(* Logix 5000 project; controller QW361 vendor 1 type 14 code 107 rev 32.11; software revision 32.00; part 10 of 20 *)

        [1241].log_data[0].time := 300.0, [1241].log_data[0].minminute := 55, [1241].log_data[0].maxminute := 55, [1241].log_data[0].valid := 1, [1241].log_data[1].valid := 1, [1241].log_data[2].valid := 1, [1241].log_data[3].valid := 1, [1241].log_data[4].valid := 1, [1241].time.Year := 2022, [1241].time.Month := 4, [1241].time.Day := 28, [1241].time.Hour := 4, [1241].time.Minute := 59, [1241].time.Second := 59, [1241].time.DST_ON := 1, [1242].log_data[0].min := 1.0, [1242].log_data[0].max := 1.0, [1242].log_data[0].total := 300.0, [1242].log_data[0].time := 300.0, [1242].log_data[0].valid := 1, [1242].log_data[1].valid := 1, [1242].log_data[2].valid := 1, [1242].log_data[3].valid := 1, [1242].log_data[4].valid := 1, [1242].time.Year := 2022, [1242].time.Month := 4, [1242].time.Day := 28, [1242].time.Hour := 5, [1242].time.Minute := 4, [1242].time.Second := 59, [1242].time.DST_ON := 1, [1243].log_data[0].min := 1.0, [1243].log_data[0].max := 1.0, [1243].log_data[0].total := 300.0, [1243].log_data[0].time := 300.0, [1243].log_data[0].minminute := 5, [1243].log_data[0].maxminute := 5, [1243].log_data[0].valid := 1, [1243].log_data[1].valid := 1, [1243].log_data[2].valid := 1, [1243].log_data[3].valid := 1, [1243].log_data[4].valid := 1, [1243].time.Year := 2022, [1243].time.Month := 4, [1243].time.Day := 28, [1243].time.Hour := 5, [1243].time.Minute := 9, [1243].time.Second := 59, [1243].time.DST_ON := 1, [1244].log_data[0].min := 1.0, [1244].log_data[0].max := 1.0, [1244].log_data[0].total := 300.0, [1244].log_data[0].time := 300.0, [1244].log_data[0].minminute := 10, [1244].log_data[0].maxminute := 10, [1244].log_data[0].valid := 1, [1244].log_data[1].valid := 1, [1244].log_data[2].valid := 1, [1244].log_data[3].valid := 1, [1244].log_data[4].valid := 1,
        [1244].time.Year := 2022, [1244].time.Month := 4, [1244].time.Day := 28, [1244].time.Hour := 5, [1244].time.Minute := 14, [1244].time.Second := 59, [1244].time.DST_ON := 1, [1245].log_data[0].min := 1.0, [1245].log_data[0].max := 1.0, [1245].log_data[0].total := 300.0, [1245].log_data[0].time := 300.0, [1245].log_data[0].minminute := 15, [1245].log_data[0].maxminute := 15, [1245].log_data[0].valid := 1, [1245].log_data[1].valid := 1, [1245].log_data[2].valid := 1, [1245].log_data[3].valid := 1, [1245].log_data[4].valid := 1, [1245].time.Year := 2022, [1245].time.Month := 4, [1245].time.Day := 28, [1245].time.Hour := 5, [1245].time.Minute := 19, [1245].time.Second := 59, [1245].time.DST_ON := 1, [1246].log_data[0].min := 1.0, [1246].log_data[0].max := 1.0, [1246].log_data[0].total := 300.0, [1246].log_data[0].time := 300.0, [1246].log_data[0].minminute := 20, [1246].log_data[0].maxminute := 20, [1246].log_data[0].valid := 1, [1246].log_data[1].valid := 1, [1246].log_data[2].valid := 1, [1246].log_data[3].valid := 1, [1246].log_data[4].valid := 1, [1246].time.Year := 2022, [1246].time.Month := 4, [1246].time.Day := 28, [1246].time.Hour := 5, [1246].time.Minute := 24, [1246].time.Second := 59, [1246].time.DST_ON := 1, [1247].log_data[0].min := 1.0, [1247].log_data[0].max := 1.0, [1247].log_data[0].total := 300.0, [1247].log_data[0].time := 300.0, [1247].log_data[0].minminute := 25, [1247].log_data[0].maxminute := 25, [1247].log_data[0].valid := 1, [1247].log_data[1].valid := 1, [1247].log_data[2].valid := 1, [1247].log_data[3].valid := 1, [1247].log_data[4].valid := 1, [1247].time.Year := 2022, [1247].time.Month := 4, [1247].time.Day := 28, [1247].time.Hour := 5, [1247].time.Minute := 29, [1247].time.Second := 59,
        [1247].time.DST_ON := 1, [1248].log_data[0].min := 1.0, [1248].log_data[0].max := 1.0, [1248].log_data[0].total := 300.0, [1248].log_data[0].time := 300.0, [1248].log_data[0].minminute := 30, [1248].log_data[0].maxminute := 30, [1248].log_data[0].valid := 1, [1248].log_data[1].valid := 1, [1248].log_data[2].valid := 1, [1248].log_data[3].valid := 1, [1248].log_data[4].valid := 1, [1248].time.Year := 2022, [1248].time.Month := 4, [1248].time.Day := 28, [1248].time.Hour := 5, [1248].time.Minute := 34, [1248].time.Second := 59, [1248].time.DST_ON := 1, [1249].log_data[0].min := 1.0, [1249].log_data[0].max := 1.0, [1249].log_data[0].total := 300.0, [1249].log_data[0].time := 300.0, [1249].log_data[0].minminute := 35, [1249].log_data[0].maxminute := 35, [1249].log_data[0].valid := 1, [1249].log_data[1].valid := 1, [1249].log_data[2].valid := 1, [1249].log_data[3].valid := 1, [1249].log_data[4].valid := 1, [1249].time.Year := 2022, [1249].time.Month := 4, [1249].time.Day := 28, [1249].time.Hour := 5, [1249].time.Minute := 39, [1249].time.Second := 59, [1249].time.DST_ON := 1, [1250].log_data[0].min := 1.0, [1250].log_data[0].max := 1.0, [1250].log_data[0].total := 300.0, [1250].log_data[0].time := 300.0, [1250].log_data[0].minminute := 40, [1250].log_data[0].maxminute := 40, [1250].log_data[0].valid := 1, [1250].log_data[1].valid := 1, [1250].log_data[2].valid := 1, [1250].log_data[3].valid := 1, [1250].log_data[4].valid := 1, [1250].time.Year := 2022, [1250].time.Month := 4, [1250].time.Day := 28, [1250].time.Hour := 5, [1250].time.Minute := 44, [1250].time.Second := 59, [1250].time.DST_ON := 1, [1251].log_data[0].min := 1.0, [1251].log_data[0].max := 1.0, [1251].log_data[0].total := 300.0, [1251].log_data[0].time := 300.0, [1251].log_data[0].minminute := 45,
        [1251].log_data[0].maxminute := 45, [1251].log_data[0].valid := 1, [1251].log_data[1].valid := 1, [1251].log_data[2].valid := 1, [1251].log_data[3].valid := 1, [1251].log_data[4].valid := 1, [1251].time.Year := 2022, [1251].time.Month := 4, [1251].time.Day := 28, [1251].time.Hour := 5, [1251].time.Minute := 49, [1251].time.Second := 59, [1251].time.DST_ON := 1, [1252].log_data[0].min := 1.0, [1252].log_data[0].max := 1.0, [1252].log_data[0].total := 300.0, [1252].log_data[0].time := 300.0, [1252].log_data[0].minminute := 50, [1252].log_data[0].maxminute := 50, [1252].log_data[0].valid := 1, [1252].log_data[1].valid := 1, [1252].log_data[2].valid := 1, [1252].log_data[3].valid := 1, [1252].log_data[4].valid := 1, [1252].time.Year := 2022, [1252].time.Month := 4, [1252].time.Day := 28, [1252].time.Hour := 5, [1252].time.Minute := 54, [1252].time.Second := 59, [1252].time.DST_ON := 1, [1253].log_data[0].min := 1.0, [1253].log_data[0].max := 1.0, [1253].log_data[0].total := 300.0, [1253].log_data[0].time := 300.0, [1253].log_data[0].minminute := 55, [1253].log_data[0].maxminute := 55, [1253].log_data[0].valid := 1, [1253].log_data[1].valid := 1, [1253].log_data[2].valid := 1, [1253].log_data[3].valid := 1, [1253].log_data[4].valid := 1, [1253].time.Year := 2022, [1253].time.Month := 4, [1253].time.Day := 28, [1253].time.Hour := 5, [1253].time.Minute := 59, [1253].time.Second := 59, [1253].time.DST_ON := 1, [1254].log_data[0].min := 1.0, [1254].log_data[0].max := 1.0, [1254].log_data[0].total := 300.0, [1254].log_data[0].time := 300.0, [1254].log_data[0].valid := 1, [1254].log_data[1].valid := 1, [1254].log_data[2].valid := 1, [1254].log_data[3].valid := 1, [1254].log_data[4].valid := 1, [1254].time.Year := 2022, [1254].time.Month := 4,
        [1254].time.Day := 28, [1254].time.Hour := 6, [1254].time.Minute := 4, [1254].time.Second := 59, [1254].time.DST_ON := 1, [1255].log_data[0].min := 1.0, [1255].log_data[0].max := 1.0, [1255].log_data[0].total := 300.0, [1255].log_data[0].time := 300.0, [1255].log_data[0].minminute := 5, [1255].log_data[0].maxminute := 5, [1255].log_data[0].valid := 1, [1255].log_data[1].valid := 1, [1255].log_data[2].valid := 1, [1255].log_data[3].valid := 1, [1255].log_data[4].valid := 1, [1255].time.Year := 2022, [1255].time.Month := 4, [1255].time.Day := 28, [1255].time.Hour := 6, [1255].time.Minute := 9, [1255].time.Second := 59, [1255].time.DST_ON := 1, [1256].log_data[0].min := 1.0, [1256].log_data[0].max := 1.0, [1256].log_data[0].total := 300.0, [1256].log_data[0].time := 300.0, [1256].log_data[0].minminute := 10, [1256].log_data[0].maxminute := 10, [1256].log_data[0].valid := 1, [1256].log_data[1].valid := 1, [1256].log_data[2].valid := 1, [1256].log_data[3].valid := 1, [1256].log_data[4].valid := 1, [1256].time.Year := 2022, [1256].time.Month := 4, [1256].time.Day := 28, [1256].time.Hour := 6, [1256].time.Minute := 14, [1256].time.Second := 59, [1256].time.DST_ON := 1, [1257].log_data[0].min := 1.0, [1257].log_data[0].max := 1.0, [1257].log_data[0].total := 299.999, [1257].log_data[0].time := 299.999, [1257].log_data[0].minminute := 15, [1257].log_data[0].maxminute := 15, [1257].log_data[0].valid := 1, [1257].log_data[1].valid := 1, [1257].log_data[2].valid := 1, [1257].log_data[3].valid := 1, [1257].log_data[4].valid := 1, [1257].time.Year := 2022, [1257].time.Month := 4, [1257].time.Day := 28, [1257].time.Hour := 6, [1257].time.Minute := 19, [1257].time.Second := 59, [1257].time.DST_ON := 1, [1258].log_data[0].min := 1.0,
        [1258].log_data[0].max := 1.0, [1258].log_data[0].total := 300.0, [1258].log_data[0].time := 300.0, [1258].log_data[0].minminute := 20, [1258].log_data[0].maxminute := 20, [1258].log_data[0].valid := 1, [1258].log_data[1].valid := 1, [1258].log_data[2].valid := 1, [1258].log_data[3].valid := 1, [1258].log_data[4].valid := 1, [1258].time.Year := 2022, [1258].time.Month := 4, [1258].time.Day := 28, [1258].time.Hour := 6, [1258].time.Minute := 24, [1258].time.Second := 59, [1258].time.DST_ON := 1, [1259].log_data[0].min := 1.0, [1259].log_data[0].max := 1.0, [1259].log_data[0].total := 300.0, [1259].log_data[0].time := 300.0, [1259].log_data[0].minminute := 25, [1259].log_data[0].maxminute := 25, [1259].log_data[0].valid := 1, [1259].log_data[1].valid := 1, [1259].log_data[2].valid := 1, [1259].log_data[3].valid := 1, [1259].log_data[4].valid := 1, [1259].time.Year := 2022, [1259].time.Month := 4, [1259].time.Day := 28, [1259].time.Hour := 6, [1259].time.Minute := 29, [1259].time.Second := 59, [1259].time.DST_ON := 1, [1260].log_data[0].min := 1.0, [1260].log_data[0].max := 1.0, [1260].log_data[0].total := 300.0, [1260].log_data[0].time := 300.0, [1260].log_data[0].minminute := 30, [1260].log_data[0].maxminute := 30, [1260].log_data[0].valid := 1, [1260].log_data[1].valid := 1, [1260].log_data[2].valid := 1, [1260].log_data[3].valid := 1, [1260].log_data[4].valid := 1, [1260].time.Year := 2022, [1260].time.Month := 4, [1260].time.Day := 28, [1260].time.Hour := 6, [1260].time.Minute := 34, [1260].time.Second := 59, [1260].time.DST_ON := 1, [1261].log_data[0].min := 1.0, [1261].log_data[0].max := 1.0, [1261].log_data[0].total := 300.0, [1261].log_data[0].time := 300.0, [1261].log_data[0].minminute := 35, [1261].log_data[0].maxminute := 35, [1261].log_data[0].valid := 1,
        [1261].log_data[1].valid := 1, [1261].log_data[2].valid := 1, [1261].log_data[3].valid := 1, [1261].log_data[4].valid := 1, [1261].time.Year := 2022, [1261].time.Month := 4, [1261].time.Day := 28, [1261].time.Hour := 6, [1261].time.Minute := 39, [1261].time.Second := 59, [1261].time.DST_ON := 1, [1262].log_data[0].min := 1.0, [1262].log_data[0].max := 1.0, [1262].log_data[0].total := 300.0, [1262].log_data[0].time := 300.0, [1262].log_data[0].minminute := 40, [1262].log_data[0].maxminute := 40, [1262].log_data[0].valid := 1, [1262].log_data[1].valid := 1, [1262].log_data[2].valid := 1, [1262].log_data[3].valid := 1, [1262].log_data[4].valid := 1, [1262].time.Year := 2022, [1262].time.Month := 4, [1262].time.Day := 28, [1262].time.Hour := 6, [1262].time.Minute := 44, [1262].time.Second := 59, [1262].time.DST_ON := 1, [1263].log_data[0].min := 1.0, [1263].log_data[0].max := 1.0, [1263].log_data[0].total := 300.0, [1263].log_data[0].time := 300.0, [1263].log_data[0].minminute := 45, [1263].log_data[0].maxminute := 45, [1263].log_data[0].valid := 1, [1263].log_data[1].valid := 1, [1263].log_data[2].valid := 1, [1263].log_data[3].valid := 1, [1263].log_data[4].valid := 1, [1263].time.Year := 2022, [1263].time.Month := 4, [1263].time.Day := 28, [1263].time.Hour := 6, [1263].time.Minute := 49, [1263].time.Second := 59, [1263].time.DST_ON := 1, [1264].log_data[0].min := 1.0, [1264].log_data[0].max := 1.0, [1264].log_data[0].total := 300.0, [1264].log_data[0].time := 300.0, [1264].log_data[0].minminute := 50, [1264].log_data[0].maxminute := 50, [1264].log_data[0].valid := 1, [1264].log_data[1].valid := 1, [1264].log_data[2].valid := 1, [1264].log_data[3].valid := 1, [1264].log_data[4].valid := 1, [1264].time.Year := 2022, [1264].time.Month := 4,
        [1264].time.Day := 28, [1264].time.Hour := 6, [1264].time.Minute := 54, [1264].time.Second := 59, [1264].time.DST_ON := 1, [1265].log_data[0].min := 1.0, [1265].log_data[0].max := 1.0, [1265].log_data[0].total := 300.0, [1265].log_data[0].time := 300.0, [1265].log_data[0].minminute := 55, [1265].log_data[0].maxminute := 55, [1265].log_data[0].valid := 1, [1265].log_data[1].valid := 1, [1265].log_data[2].valid := 1, [1265].log_data[3].valid := 1, [1265].log_data[4].valid := 1, [1265].time.Year := 2022, [1265].time.Month := 4, [1265].time.Day := 28, [1265].time.Hour := 6, [1265].time.Minute := 59, [1265].time.Second := 59, [1265].time.DST_ON := 1, [1266].log_data[0].min := 1.0, [1266].log_data[0].max := 1.0, [1266].log_data[0].total := 300.0, [1266].log_data[0].time := 300.0, [1266].log_data[0].valid := 1, [1266].log_data[1].valid := 1, [1266].log_data[2].valid := 1, [1266].log_data[3].valid := 1, [1266].log_data[4].valid := 1, [1266].time.Year := 2022, [1266].time.Month := 4, [1266].time.Day := 28, [1266].time.Hour := 7, [1266].time.Minute := 4, [1266].time.Second := 59, [1266].time.DST_ON := 1, [1267].log_data[0].min := 1.0, [1267].log_data[0].max := 1.0, [1267].log_data[0].total := 300.0, [1267].log_data[0].time := 300.0, [1267].log_data[0].minminute := 5, [1267].log_data[0].maxminute := 5, [1267].log_data[0].valid := 1, [1267].log_data[1].valid := 1, [1267].log_data[2].valid := 1, [1267].log_data[3].valid := 1, [1267].log_data[4].valid := 1, [1267].time.Year := 2022, [1267].time.Month := 4, [1267].time.Day := 28, [1267].time.Hour := 7, [1267].time.Minute := 9, [1267].time.Second := 59, [1267].time.DST_ON := 1, [1268].log_data[0].min := 1.0, [1268].log_data[0].max := 1.0, [1268].log_data[0].total := 300.0,
        [1268].log_data[0].time := 300.0, [1268].log_data[0].minminute := 10, [1268].log_data[0].maxminute := 10, [1268].log_data[0].valid := 1, [1268].log_data[1].valid := 1, [1268].log_data[2].valid := 1, [1268].log_data[3].valid := 1, [1268].log_data[4].valid := 1, [1268].time.Year := 2022, [1268].time.Month := 4, [1268].time.Day := 28, [1268].time.Hour := 7, [1268].time.Minute := 14, [1268].time.Second := 59, [1268].time.DST_ON := 1, [1269].log_data[0].min := 1.0, [1269].log_data[0].max := 1.0, [1269].log_data[0].total := 300.0, [1269].log_data[0].time := 300.0, [1269].log_data[0].minminute := 15, [1269].log_data[0].maxminute := 15, [1269].log_data[0].valid := 1, [1269].log_data[1].valid := 1, [1269].log_data[2].valid := 1, [1269].log_data[3].valid := 1, [1269].log_data[4].valid := 1, [1269].time.Year := 2022, [1269].time.Month := 4, [1269].time.Day := 28, [1269].time.Hour := 7, [1269].time.Minute := 19, [1269].time.Second := 59, [1269].time.DST_ON := 1, [1270].log_data[0].min := 1.0, [1270].log_data[0].max := 1.0, [1270].log_data[0].total := 300.0, [1270].log_data[0].time := 300.0, [1270].log_data[0].minminute := 20, [1270].log_data[0].maxminute := 20, [1270].log_data[0].valid := 1, [1270].log_data[1].valid := 1, [1270].log_data[2].valid := 1, [1270].log_data[3].valid := 1, [1270].log_data[4].valid := 1, [1270].time.Year := 2022, [1270].time.Month := 4, [1270].time.Day := 28, [1270].time.Hour := 7, [1270].time.Minute := 24, [1270].time.Second := 59, [1270].time.DST_ON := 1, [1271].log_data[0].min := 1.0, [1271].log_data[0].max := 1.0, [1271].log_data[0].total := 300.0, [1271].log_data[0].time := 300.0, [1271].log_data[0].minminute := 25, [1271].log_data[0].maxminute := 25, [1271].log_data[0].valid := 1, [1271].log_data[1].valid := 1, [1271].log_data[2].valid := 1,
        [1271].log_data[3].valid := 1, [1271].log_data[4].valid := 1, [1271].time.Year := 2022, [1271].time.Month := 4, [1271].time.Day := 28, [1271].time.Hour := 7, [1271].time.Minute := 29, [1271].time.Second := 59, [1271].time.DST_ON := 1, [1272].log_data[0].min := 1.0, [1272].log_data[0].max := 1.0, [1272].log_data[0].total := 300.0, [1272].log_data[0].time := 300.0, [1272].log_data[0].minminute := 30, [1272].log_data[0].maxminute := 30, [1272].log_data[0].valid := 1, [1272].log_data[1].valid := 1, [1272].log_data[2].valid := 1, [1272].log_data[3].valid := 1, [1272].log_data[4].valid := 1, [1272].time.Year := 2022, [1272].time.Month := 4, [1272].time.Day := 28, [1272].time.Hour := 7, [1272].time.Minute := 34, [1272].time.Second := 59, [1272].time.DST_ON := 1, [1273].log_data[0].min := 1.0, [1273].log_data[0].max := 1.0, [1273].log_data[0].total := 300.0, [1273].log_data[0].time := 300.0, [1273].log_data[0].minminute := 35, [1273].log_data[0].maxminute := 35, [1273].log_data[0].valid := 1, [1273].log_data[1].valid := 1, [1273].log_data[2].valid := 1, [1273].log_data[3].valid := 1, [1273].log_data[4].valid := 1, [1273].time.Year := 2022, [1273].time.Month := 4, [1273].time.Day := 28, [1273].time.Hour := 7, [1273].time.Minute := 39, [1273].time.Second := 59, [1273].time.DST_ON := 1, [1274].log_data[0].min := 1.0, [1274].log_data[0].max := 1.0, [1274].log_data[0].total := 300.0, [1274].log_data[0].time := 300.0, [1274].log_data[0].minminute := 40, [1274].log_data[0].maxminute := 40, [1274].log_data[0].valid := 1, [1274].log_data[1].valid := 1, [1274].log_data[2].valid := 1, [1274].log_data[3].valid := 1, [1274].log_data[4].valid := 1, [1274].time.Year := 2022, [1274].time.Month := 4, [1274].time.Day := 28, [1274].time.Hour := 7,
        [1274].time.Minute := 44, [1274].time.Second := 59, [1274].time.DST_ON := 1, [1275].log_data[0].min := 1.0, [1275].log_data[0].max := 1.0, [1275].log_data[0].total := 300.0, [1275].log_data[0].time := 300.0, [1275].log_data[0].minminute := 45, [1275].log_data[0].maxminute := 45, [1275].log_data[0].valid := 1, [1275].log_data[1].valid := 1, [1275].log_data[2].valid := 1, [1275].log_data[3].valid := 1, [1275].log_data[4].valid := 1, [1275].time.Year := 2022, [1275].time.Month := 4, [1275].time.Day := 28, [1275].time.Hour := 7, [1275].time.Minute := 49, [1275].time.Second := 59, [1275].time.DST_ON := 1, [1276].log_data[0].min := 1.0, [1276].log_data[0].max := 1.0, [1276].log_data[0].total := 300.0, [1276].log_data[0].time := 300.0, [1276].log_data[0].minminute := 50, [1276].log_data[0].maxminute := 50, [1276].log_data[0].valid := 1, [1276].log_data[1].valid := 1, [1276].log_data[2].valid := 1, [1276].log_data[3].valid := 1, [1276].log_data[4].valid := 1, [1276].time.Year := 2022, [1276].time.Month := 4, [1276].time.Day := 28, [1276].time.Hour := 7, [1276].time.Minute := 54, [1276].time.Second := 59, [1276].time.DST_ON := 1, [1277].log_data[0].min := 1.0, [1277].log_data[0].max := 1.0, [1277].log_data[0].total := 300.0, [1277].log_data[0].time := 300.0, [1277].log_data[0].minminute := 55, [1277].log_data[0].maxminute := 55, [1277].log_data[0].valid := 1, [1277].log_data[1].valid := 1, [1277].log_data[2].valid := 1, [1277].log_data[3].valid := 1, [1277].log_data[4].valid := 1, [1277].time.Year := 2022, [1277].time.Month := 4, [1277].time.Day := 28, [1277].time.Hour := 7, [1277].time.Minute := 59, [1277].time.Second := 59, [1277].time.DST_ON := 1, [1278].log_data[0].min := 1.0, [1278].log_data[0].max := 1.0, [1278].log_data[0].total := 300.0,
        [1278].log_data[0].time := 300.0, [1278].log_data[0].valid := 1, [1278].log_data[1].valid := 1, [1278].log_data[2].valid := 1, [1278].log_data[3].valid := 1, [1278].log_data[4].valid := 1, [1278].time.Year := 2022, [1278].time.Month := 4, [1278].time.Day := 28, [1278].time.Hour := 8, [1278].time.Minute := 4, [1278].time.Second := 59, [1278].time.DST_ON := 1, [1279].log_data[0].min := 1.0, [1279].log_data[0].max := 1.0, [1279].log_data[0].total := 300.0, [1279].log_data[0].time := 300.0, [1279].log_data[0].minminute := 5, [1279].log_data[0].maxminute := 5, [1279].log_data[0].valid := 1, [1279].log_data[1].valid := 1, [1279].log_data[2].valid := 1, [1279].log_data[3].valid := 1, [1279].log_data[4].valid := 1, [1279].time.Year := 2022, [1279].time.Month := 4, [1279].time.Day := 28, [1279].time.Hour := 8, [1279].time.Minute := 9, [1279].time.Second := 59, [1279].time.DST_ON := 1, [1280].log_data[0].min := 1.0, [1280].log_data[0].max := 1.0, [1280].log_data[0].total := 300.0, [1280].log_data[0].time := 300.0, [1280].log_data[0].minminute := 10, [1280].log_data[0].maxminute := 10, [1280].log_data[0].valid := 1, [1280].log_data[1].valid := 1, [1280].log_data[2].valid := 1, [1280].log_data[3].valid := 1, [1280].log_data[4].valid := 1, [1280].time.Year := 2022, [1280].time.Month := 4, [1280].time.Day := 28, [1280].time.Hour := 8, [1280].time.Minute := 14, [1280].time.Second := 59, [1280].time.DST_ON := 1, [1281].log_data[0].min := 1.0, [1281].log_data[0].max := 1.0, [1281].log_data[0].total := 300.0, [1281].log_data[0].time := 300.0, [1281].log_data[0].minminute := 15, [1281].log_data[0].maxminute := 15, [1281].log_data[0].valid := 1, [1281].log_data[1].valid := 1, [1281].log_data[2].valid := 1, [1281].log_data[3].valid := 1, [1281].log_data[4].valid := 1,
        [1281].time.Year := 2022, [1281].time.Month := 4, [1281].time.Day := 28, [1281].time.Hour := 8, [1281].time.Minute := 19, [1281].time.Second := 59, [1281].time.DST_ON := 1, [1282].log_data[0].min := 1.0, [1282].log_data[0].max := 1.0, [1282].log_data[0].total := 300.0, [1282].log_data[0].time := 300.0, [1282].log_data[0].minminute := 20, [1282].log_data[0].maxminute := 20, [1282].log_data[0].valid := 1, [1282].log_data[1].valid := 1, [1282].log_data[2].valid := 1, [1282].log_data[3].valid := 1, [1282].log_data[4].valid := 1, [1282].time.Year := 2022, [1282].time.Month := 4, [1282].time.Day := 28, [1282].time.Hour := 8, [1282].time.Minute := 24, [1282].time.Second := 59, [1282].time.DST_ON := 1, [1283].log_data[0].min := 1.0, [1283].log_data[0].max := 1.0, [1283].log_data[0].total := 300.0, [1283].log_data[0].time := 300.0, [1283].log_data[0].minminute := 25, [1283].log_data[0].maxminute := 25, [1283].log_data[0].valid := 1, [1283].log_data[1].valid := 1, [1283].log_data[2].valid := 1, [1283].log_data[3].valid := 1, [1283].log_data[4].valid := 1, [1283].time.Year := 2022, [1283].time.Month := 4, [1283].time.Day := 28, [1283].time.Hour := 8, [1283].time.Minute := 29, [1283].time.Second := 59, [1283].time.DST_ON := 1, [1284].log_data[0].min := 1.0, [1284].log_data[0].max := 1.0, [1284].log_data[0].total := 300.0, [1284].log_data[0].time := 300.0, [1284].log_data[0].minminute := 30, [1284].log_data[0].maxminute := 30, [1284].log_data[0].valid := 1, [1284].log_data[1].valid := 1, [1284].log_data[2].valid := 1, [1284].log_data[3].valid := 1, [1284].log_data[4].valid := 1, [1284].time.Year := 2022, [1284].time.Month := 4, [1284].time.Day := 28, [1284].time.Hour := 8, [1284].time.Minute := 34, [1284].time.Second := 59,
        [1284].time.DST_ON := 1, [1285].log_data[0].min := 1.0, [1285].log_data[0].max := 1.0, [1285].log_data[0].total := 300.0, [1285].log_data[0].time := 300.0, [1285].log_data[0].minminute := 35, [1285].log_data[0].maxminute := 35, [1285].log_data[0].valid := 1, [1285].log_data[1].valid := 1, [1285].log_data[2].valid := 1, [1285].log_data[3].valid := 1, [1285].log_data[4].valid := 1, [1285].time.Year := 2022, [1285].time.Month := 4, [1285].time.Day := 28, [1285].time.Hour := 8, [1285].time.Minute := 39, [1285].time.Second := 59, [1285].time.DST_ON := 1, [1286].log_data[0].min := 1.0, [1286].log_data[0].max := 1.0, [1286].log_data[0].total := 300.0, [1286].log_data[0].time := 300.0, [1286].log_data[0].minminute := 40, [1286].log_data[0].maxminute := 40, [1286].log_data[0].valid := 1, [1286].log_data[1].valid := 1, [1286].log_data[2].valid := 1, [1286].log_data[3].valid := 1, [1286].log_data[4].valid := 1, [1286].time.Year := 2022, [1286].time.Month := 4, [1286].time.Day := 28, [1286].time.Hour := 8, [1286].time.Minute := 44, [1286].time.Second := 59, [1286].time.DST_ON := 1, [1287].log_data[0].min := 1.0, [1287].log_data[0].max := 1.0, [1287].log_data[0].total := 300.0, [1287].log_data[0].time := 300.0, [1287].log_data[0].minminute := 45, [1287].log_data[0].maxminute := 45, [1287].log_data[0].valid := 1, [1287].log_data[1].valid := 1, [1287].log_data[2].valid := 1, [1287].log_data[3].valid := 1, [1287].log_data[4].valid := 1, [1287].time.Year := 2022, [1287].time.Month := 4, [1287].time.Day := 28, [1287].time.Hour := 8, [1287].time.Minute := 49, [1287].time.Second := 59, [1287].time.DST_ON := 1, [1288].log_data[0].min := 1.0, [1288].log_data[0].max := 1.0, [1288].log_data[0].total := 300.0, [1288].log_data[0].time := 300.0, [1288].log_data[0].minminute := 50,
        [1288].log_data[0].maxminute := 50, [1288].log_data[0].valid := 1, [1288].log_data[1].valid := 1, [1288].log_data[2].valid := 1, [1288].log_data[3].valid := 1, [1288].log_data[4].valid := 1, [1288].time.Year := 2022, [1288].time.Month := 4, [1288].time.Day := 28, [1288].time.Hour := 8, [1288].time.Minute := 54, [1288].time.Second := 59, [1288].time.DST_ON := 1, [1289].log_data[0].min := 1.0, [1289].log_data[0].max := 1.0, [1289].log_data[0].total := 300.0, [1289].log_data[0].time := 300.0, [1289].log_data[0].minminute := 55, [1289].log_data[0].maxminute := 55, [1289].log_data[0].valid := 1, [1289].log_data[1].valid := 1, [1289].log_data[2].valid := 1, [1289].log_data[3].valid := 1, [1289].log_data[4].valid := 1, [1289].time.Year := 2022, [1289].time.Month := 4, [1289].time.Day := 28, [1289].time.Hour := 8, [1289].time.Minute := 59, [1289].time.Second := 59, [1289].time.DST_ON := 1, [1290].log_data[0].min := 1.0, [1290].log_data[0].max := 1.0, [1290].log_data[0].total := 300.0, [1290].log_data[0].time := 300.0, [1290].log_data[0].valid := 1, [1290].log_data[1].valid := 1, [1290].log_data[2].valid := 1, [1290].log_data[3].valid := 1, [1290].log_data[4].valid := 1, [1290].time.Year := 2022, [1290].time.Month := 4, [1290].time.Day := 28, [1290].time.Hour := 9, [1290].time.Minute := 4, [1290].time.Second := 59, [1290].time.DST_ON := 1, [1291].log_data[0].min := 1.0, [1291].log_data[0].max := 1.0, [1291].log_data[0].total := 300.0, [1291].log_data[0].time := 300.0, [1291].log_data[0].minminute := 5, [1291].log_data[0].maxminute := 5, [1291].log_data[0].valid := 1, [1291].log_data[1].valid := 1, [1291].log_data[2].valid := 1, [1291].log_data[3].valid := 1, [1291].log_data[4].valid := 1, [1291].time.Year := 2022, [1291].time.Month := 4,
        [1291].time.Day := 28, [1291].time.Hour := 9, [1291].time.Minute := 9, [1291].time.Second := 59, [1291].time.DST_ON := 1, [1292].log_data[0].min := 1.0, [1292].log_data[0].max := 1.0, [1292].log_data[0].total := 300.0, [1292].log_data[0].time := 300.0, [1292].log_data[0].minminute := 10, [1292].log_data[0].maxminute := 10, [1292].log_data[0].valid := 1, [1292].log_data[1].valid := 1, [1292].log_data[2].valid := 1, [1292].log_data[3].valid := 1, [1292].log_data[4].valid := 1, [1292].time.Year := 2022, [1292].time.Month := 4, [1292].time.Day := 28, [1292].time.Hour := 9, [1292].time.Minute := 14, [1292].time.Second := 59, [1292].time.DST_ON := 1, [1293].log_data[0].min := 1.0, [1293].log_data[0].max := 1.0, [1293].log_data[0].total := 300.0, [1293].log_data[0].time := 300.0, [1293].log_data[0].minminute := 15, [1293].log_data[0].maxminute := 15, [1293].log_data[0].valid := 1, [1293].log_data[1].valid := 1, [1293].log_data[2].valid := 1, [1293].log_data[3].valid := 1, [1293].log_data[4].valid := 1, [1293].time.Year := 2022, [1293].time.Month := 4, [1293].time.Day := 28, [1293].time.Hour := 9, [1293].time.Minute := 19, [1293].time.Second := 59, [1293].time.DST_ON := 1, [1294].log_data[0].min := 1.0, [1294].log_data[0].max := 1.0, [1294].log_data[0].total := 300.0, [1294].log_data[0].time := 300.0, [1294].log_data[0].minminute := 20, [1294].log_data[0].maxminute := 20, [1294].log_data[0].valid := 1, [1294].log_data[1].valid := 1, [1294].log_data[2].valid := 1, [1294].log_data[3].valid := 1, [1294].log_data[4].valid := 1, [1294].time.Year := 2022, [1294].time.Month := 4, [1294].time.Day := 28, [1294].time.Hour := 9, [1294].time.Minute := 24, [1294].time.Second := 59, [1294].time.DST_ON := 1, [1295].log_data[0].min := 1.0,
        [1295].log_data[0].max := 1.0, [1295].log_data[0].total := 300.0, [1295].log_data[0].time := 300.0, [1295].log_data[0].minminute := 25, [1295].log_data[0].maxminute := 25, [1295].log_data[0].valid := 1, [1295].log_data[1].valid := 1, [1295].log_data[2].valid := 1, [1295].log_data[3].valid := 1, [1295].log_data[4].valid := 1, [1295].time.Year := 2022, [1295].time.Month := 4, [1295].time.Day := 28, [1295].time.Hour := 9, [1295].time.Minute := 29, [1295].time.Second := 59, [1295].time.DST_ON := 1, [1296].log_data[0].min := 1.0, [1296].log_data[0].max := 1.0, [1296].log_data[0].total := 300.0, [1296].log_data[0].time := 300.0, [1296].log_data[0].minminute := 30, [1296].log_data[0].maxminute := 30, [1296].log_data[0].valid := 1, [1296].log_data[1].valid := 1, [1296].log_data[2].valid := 1, [1296].log_data[3].valid := 1, [1296].log_data[4].valid := 1, [1296].time.Year := 2022, [1296].time.Month := 4, [1296].time.Day := 28, [1296].time.Hour := 9, [1296].time.Minute := 34, [1296].time.Second := 59, [1296].time.DST_ON := 1, [1297].log_data[0].min := 1.0, [1297].log_data[0].max := 1.0, [1297].log_data[0].total := 300.0, [1297].log_data[0].time := 300.0, [1297].log_data[0].minminute := 35, [1297].log_data[0].maxminute := 35, [1297].log_data[0].valid := 1, [1297].log_data[1].valid := 1, [1297].log_data[2].valid := 1, [1297].log_data[3].valid := 1, [1297].log_data[4].valid := 1, [1297].time.Year := 2022, [1297].time.Month := 4, [1297].time.Day := 28, [1297].time.Hour := 9, [1297].time.Minute := 39, [1297].time.Second := 59, [1297].time.DST_ON := 1, [1298].log_data[0].min := 1.0, [1298].log_data[0].max := 1.0, [1298].log_data[0].total := 300.0, [1298].log_data[0].time := 300.0, [1298].log_data[0].minminute := 40, [1298].log_data[0].maxminute := 40, [1298].log_data[0].valid := 1,
        [1298].log_data[1].valid := 1, [1298].log_data[2].valid := 1, [1298].log_data[3].valid := 1, [1298].log_data[4].valid := 1, [1298].time.Year := 2022, [1298].time.Month := 4, [1298].time.Day := 28, [1298].time.Hour := 9, [1298].time.Minute := 44, [1298].time.Second := 59, [1298].time.DST_ON := 1, [1299].log_data[0].min := 1.0, [1299].log_data[0].max := 1.0, [1299].log_data[0].total := 300.0, [1299].log_data[0].time := 300.0, [1299].log_data[0].minminute := 45, [1299].log_data[0].maxminute := 45, [1299].log_data[0].valid := 1, [1299].log_data[1].valid := 1, [1299].log_data[2].valid := 1, [1299].log_data[3].valid := 1, [1299].log_data[4].valid := 1, [1299].time.Year := 2022, [1299].time.Month := 4, [1299].time.Day := 28, [1299].time.Hour := 9, [1299].time.Minute := 49, [1299].time.Second := 59, [1299].time.DST_ON := 1, [1300].log_data[0].min := 1.0, [1300].log_data[0].max := 1.0, [1300].log_data[0].total := 300.0, [1300].log_data[0].time := 300.0, [1300].log_data[0].minminute := 50, [1300].log_data[0].maxminute := 50, [1300].log_data[0].valid := 1, [1300].log_data[1].valid := 1, [1300].log_data[2].valid := 1, [1300].log_data[3].valid := 1, [1300].log_data[4].valid := 1, [1300].time.Year := 2022, [1300].time.Month := 4, [1300].time.Day := 28, [1300].time.Hour := 9, [1300].time.Minute := 54, [1300].time.Second := 59, [1300].time.DST_ON := 1, [1301].log_data[0].min := 1.0, [1301].log_data[0].max := 1.0, [1301].log_data[0].total := 300.0, [1301].log_data[0].time := 300.0, [1301].log_data[0].minminute := 55, [1301].log_data[0].maxminute := 55, [1301].log_data[0].valid := 1, [1301].log_data[1].valid := 1, [1301].log_data[2].valid := 1, [1301].log_data[3].valid := 1, [1301].log_data[4].valid := 1, [1301].time.Year := 2022, [1301].time.Month := 4,
        [1301].time.Day := 28, [1301].time.Hour := 9, [1301].time.Minute := 59, [1301].time.Second := 59, [1301].time.DST_ON := 1, [1302].log_data[0].min := 1.0, [1302].log_data[0].max := 1.0, [1302].log_data[0].total := 300.0, [1302].log_data[0].time := 300.0, [1302].log_data[0].valid := 1, [1302].log_data[1].valid := 1, [1302].log_data[2].valid := 1, [1302].log_data[3].valid := 1, [1302].log_data[4].valid := 1, [1302].time.Year := 2022, [1302].time.Month := 4, [1302].time.Day := 28, [1302].time.Hour := 10, [1302].time.Minute := 4, [1302].time.Second := 59, [1302].time.DST_ON := 1, [1303].log_data[0].min := 1.0, [1303].log_data[0].max := 1.0, [1303].log_data[0].total := 300.0, [1303].log_data[0].time := 300.0, [1303].log_data[0].minminute := 5, [1303].log_data[0].maxminute := 5, [1303].log_data[0].valid := 1, [1303].log_data[1].valid := 1, [1303].log_data[2].valid := 1, [1303].log_data[3].valid := 1, [1303].log_data[4].valid := 1, [1303].time.Year := 2022, [1303].time.Month := 4, [1303].time.Day := 28, [1303].time.Hour := 10, [1303].time.Minute := 9, [1303].time.Second := 59, [1303].time.DST_ON := 1, [1304].log_data[0].min := 1.0, [1304].log_data[0].max := 1.0, [1304].log_data[0].total := 300.0, [1304].log_data[0].time := 300.0, [1304].log_data[0].minminute := 10, [1304].log_data[0].maxminute := 10, [1304].log_data[0].valid := 1, [1304].log_data[1].valid := 1, [1304].log_data[2].valid := 1, [1304].log_data[3].valid := 1, [1304].log_data[4].valid := 1, [1304].time.Year := 2022, [1304].time.Month := 4, [1304].time.Day := 28, [1304].time.Hour := 10, [1304].time.Minute := 14, [1304].time.Second := 59, [1304].time.DST_ON := 1, [1305].log_data[0].min := 1.0, [1305].log_data[0].max := 1.0, [1305].log_data[0].total := 300.0,
        [1305].log_data[0].time := 300.0, [1305].log_data[0].minminute := 15, [1305].log_data[0].maxminute := 15, [1305].log_data[0].valid := 1, [1305].log_data[1].valid := 1, [1305].log_data[2].valid := 1, [1305].log_data[3].valid := 1, [1305].log_data[4].valid := 1, [1305].time.Year := 2022, [1305].time.Month := 4, [1305].time.Day := 28, [1305].time.Hour := 10, [1305].time.Minute := 19, [1305].time.Second := 59, [1305].time.DST_ON := 1, [1306].log_data[0].min := 1.0, [1306].log_data[0].max := 1.0, [1306].log_data[0].total := 300.0, [1306].log_data[0].time := 300.0, [1306].log_data[0].minminute := 20, [1306].log_data[0].maxminute := 20, [1306].log_data[0].valid := 1, [1306].log_data[1].valid := 1, [1306].log_data[2].valid := 1, [1306].log_data[3].valid := 1, [1306].log_data[4].valid := 1, [1306].time.Year := 2022, [1306].time.Month := 4, [1306].time.Day := 28, [1306].time.Hour := 10, [1306].time.Minute := 24, [1306].time.Second := 59, [1306].time.DST_ON := 1, [1307].log_data[0].min := 1.0, [1307].log_data[0].max := 1.0, [1307].log_data[0].total := 300.0, [1307].log_data[0].time := 300.0, [1307].log_data[0].minminute := 25, [1307].log_data[0].maxminute := 25, [1307].log_data[0].valid := 1, [1307].log_data[1].valid := 1, [1307].log_data[2].valid := 1, [1307].log_data[3].valid := 1, [1307].log_data[4].valid := 1, [1307].time.Year := 2022, [1307].time.Month := 4, [1307].time.Day := 28, [1307].time.Hour := 10, [1307].time.Minute := 29, [1307].time.Second := 59, [1307].time.DST_ON := 1, [1308].log_data[0].min := 1.0, [1308].log_data[0].max := 1.0, [1308].log_data[0].total := 300.0, [1308].log_data[0].time := 300.0, [1308].log_data[0].minminute := 30, [1308].log_data[0].maxminute := 30, [1308].log_data[0].valid := 1, [1308].log_data[1].valid := 1, [1308].log_data[2].valid := 1,
        [1308].log_data[3].valid := 1, [1308].log_data[4].valid := 1, [1308].time.Year := 2022, [1308].time.Month := 4, [1308].time.Day := 28, [1308].time.Hour := 10, [1308].time.Minute := 34, [1308].time.Second := 59, [1308].time.DST_ON := 1, [1309].log_data[0].min := 1.0, [1309].log_data[0].max := 1.0, [1309].log_data[0].total := 300.0, [1309].log_data[0].time := 300.0, [1309].log_data[0].minminute := 35, [1309].log_data[0].maxminute := 35, [1309].log_data[0].valid := 1, [1309].log_data[1].valid := 1, [1309].log_data[2].valid := 1, [1309].log_data[3].valid := 1, [1309].log_data[4].valid := 1, [1309].time.Year := 2022, [1309].time.Month := 4, [1309].time.Day := 28, [1309].time.Hour := 10, [1309].time.Minute := 39, [1309].time.Second := 59, [1309].time.DST_ON := 1, [1310].log_data[0].min := 1.0, [1310].log_data[0].max := 1.0, [1310].log_data[0].total := 300.0, [1310].log_data[0].time := 300.0, [1310].log_data[0].minminute := 40, [1310].log_data[0].maxminute := 40, [1310].log_data[0].valid := 1, [1310].log_data[1].valid := 1, [1310].log_data[2].valid := 1, [1310].log_data[3].valid := 1, [1310].log_data[4].valid := 1, [1310].time.Year := 2022, [1310].time.Month := 4, [1310].time.Day := 28, [1310].time.Hour := 10, [1310].time.Minute := 44, [1310].time.Second := 59, [1310].time.DST_ON := 1, [1311].log_data[0].min := 1.0, [1311].log_data[0].max := 1.0, [1311].log_data[0].total := 299.999, [1311].log_data[0].time := 299.999, [1311].log_data[0].minminute := 45, [1311].log_data[0].maxminute := 45, [1311].log_data[0].valid := 1, [1311].log_data[1].valid := 1, [1311].log_data[2].valid := 1, [1311].log_data[3].valid := 1, [1311].log_data[4].valid := 1, [1311].time.Year := 2022, [1311].time.Month := 4, [1311].time.Day := 28, [1311].time.Hour := 10,
        [1311].time.Minute := 49, [1311].time.Second := 59, [1311].time.DST_ON := 1, [1312].log_data[0].min := 1.0, [1312].log_data[0].max := 1.0, [1312].log_data[0].total := 300.0, [1312].log_data[0].time := 300.0, [1312].log_data[0].minminute := 50, [1312].log_data[0].maxminute := 50, [1312].log_data[0].valid := 1, [1312].log_data[1].valid := 1, [1312].log_data[2].valid := 1, [1312].log_data[3].valid := 1, [1312].log_data[4].valid := 1, [1312].time.Year := 2022, [1312].time.Month := 4, [1312].time.Day := 28, [1312].time.Hour := 10, [1312].time.Minute := 54, [1312].time.Second := 59, [1312].time.DST_ON := 1, [1313].log_data[0].min := 1.0, [1313].log_data[0].max := 1.0, [1313].log_data[0].total := 300.0, [1313].log_data[0].time := 300.0, [1313].log_data[0].minminute := 55, [1313].log_data[0].maxminute := 55, [1313].log_data[0].valid := 1, [1313].log_data[1].valid := 1, [1313].log_data[2].valid := 1, [1313].log_data[3].valid := 1, [1313].log_data[4].valid := 1, [1313].time.Year := 2022, [1313].time.Month := 4, [1313].time.Day := 28, [1313].time.Hour := 10, [1313].time.Minute := 59, [1313].time.Second := 59, [1313].time.DST_ON := 1, [1314].log_data[0].min := 1.0, [1314].log_data[0].max := 1.0, [1314].log_data[0].total := 300.0, [1314].log_data[0].time := 300.0, [1314].log_data[0].valid := 1, [1314].log_data[1].valid := 1, [1314].log_data[2].valid := 1, [1314].log_data[3].valid := 1, [1314].log_data[4].valid := 1, [1314].time.Year := 2022, [1314].time.Month := 4, [1314].time.Day := 28, [1314].time.Hour := 11, [1314].time.Minute := 4, [1314].time.Second := 59, [1314].time.DST_ON := 1, [1315].log_data[0].min := 1.0, [1315].log_data[0].max := 1.0, [1315].log_data[0].total := 300.0, [1315].log_data[0].time := 300.0, [1315].log_data[0].minminute := 5,
        [1315].log_data[0].maxminute := 5, [1315].log_data[0].valid := 1, [1315].log_data[1].valid := 1, [1315].log_data[2].valid := 1, [1315].log_data[3].valid := 1, [1315].log_data[4].valid := 1, [1315].time.Year := 2022, [1315].time.Month := 4, [1315].time.Day := 28, [1315].time.Hour := 11, [1315].time.Minute := 9, [1315].time.Second := 59, [1315].time.DST_ON := 1, [1316].log_data[0].min := 1.0, [1316].log_data[0].max := 1.0, [1316].log_data[0].total := 300.0, [1316].log_data[0].time := 300.0, [1316].log_data[0].minminute := 10, [1316].log_data[0].maxminute := 10, [1316].log_data[0].valid := 1, [1316].log_data[1].valid := 1, [1316].log_data[2].valid := 1, [1316].log_data[3].valid := 1, [1316].log_data[4].valid := 1, [1316].time.Year := 2022, [1316].time.Month := 4, [1316].time.Day := 28, [1316].time.Hour := 11, [1316].time.Minute := 14, [1316].time.Second := 59, [1316].time.DST_ON := 1, [1317].log_data[0].min := 1.0, [1317].log_data[0].max := 1.0, [1317].log_data[0].total := 300.0, [1317].log_data[0].time := 300.0, [1317].log_data[0].minminute := 15, [1317].log_data[0].maxminute := 15, [1317].log_data[0].valid := 1, [1317].log_data[1].valid := 1, [1317].log_data[2].valid := 1, [1317].log_data[3].valid := 1, [1317].log_data[4].valid := 1, [1317].time.Year := 2022, [1317].time.Month := 4, [1317].time.Day := 28, [1317].time.Hour := 11, [1317].time.Minute := 19, [1317].time.Second := 59, [1317].time.DST_ON := 1, [1318].log_data[0].min := 1.0, [1318].log_data[0].max := 1.0, [1318].log_data[0].total := 300.0, [1318].log_data[0].time := 300.0, [1318].log_data[0].minminute := 20, [1318].log_data[0].maxminute := 20, [1318].log_data[0].valid := 1, [1318].log_data[1].valid := 1, [1318].log_data[2].valid := 1, [1318].log_data[3].valid := 1, [1318].log_data[4].valid := 1,
        [1318].time.Year := 2022, [1318].time.Month := 4, [1318].time.Day := 28, [1318].time.Hour := 11, [1318].time.Minute := 24, [1318].time.Second := 59, [1318].time.DST_ON := 1, [1319].log_data[0].min := 1.0, [1319].log_data[0].max := 1.0, [1319].log_data[0].total := 300.0, [1319].log_data[0].time := 300.0, [1319].log_data[0].minminute := 25, [1319].log_data[0].maxminute := 25, [1319].log_data[0].valid := 1, [1319].log_data[1].valid := 1, [1319].log_data[2].valid := 1, [1319].log_data[3].valid := 1, [1319].log_data[4].valid := 1, [1319].time.Year := 2022, [1319].time.Month := 4, [1319].time.Day := 28, [1319].time.Hour := 11, [1319].time.Minute := 29, [1319].time.Second := 59, [1319].time.DST_ON := 1, [1320].log_data[0].min := 1.0, [1320].log_data[0].max := 1.0, [1320].log_data[0].total := 300.0, [1320].log_data[0].time := 300.0, [1320].log_data[0].minminute := 30, [1320].log_data[0].maxminute := 30, [1320].log_data[0].valid := 1, [1320].log_data[1].valid := 1, [1320].log_data[2].valid := 1, [1320].log_data[3].valid := 1, [1320].log_data[4].valid := 1, [1320].time.Year := 2022, [1320].time.Month := 4, [1320].time.Day := 28, [1320].time.Hour := 11, [1320].time.Minute := 34, [1320].time.Second := 59, [1320].time.DST_ON := 1, [1321].log_data[0].min := 1.0, [1321].log_data[0].max := 1.0, [1321].log_data[0].total := 300.0, [1321].log_data[0].time := 300.0, [1321].log_data[0].minminute := 35, [1321].log_data[0].maxminute := 35, [1321].log_data[0].valid := 1, [1321].log_data[1].valid := 1, [1321].log_data[2].valid := 1, [1321].log_data[3].valid := 1, [1321].log_data[4].valid := 1, [1321].time.Year := 2022, [1321].time.Month := 4, [1321].time.Day := 28, [1321].time.Hour := 11, [1321].time.Minute := 39, [1321].time.Second := 59,
        [1321].time.DST_ON := 1, [1322].log_data[0].min := 1.0, [1322].log_data[0].max := 1.0, [1322].log_data[0].total := 300.0, [1322].log_data[0].time := 300.0, [1322].log_data[0].minminute := 40, [1322].log_data[0].maxminute := 40, [1322].log_data[0].valid := 1, [1322].log_data[1].valid := 1, [1322].log_data[2].valid := 1, [1322].log_data[3].valid := 1, [1322].log_data[4].valid := 1, [1322].time.Year := 2022, [1322].time.Month := 4, [1322].time.Day := 28, [1322].time.Hour := 11, [1322].time.Minute := 44, [1322].time.Second := 59, [1322].time.DST_ON := 1, [1323].log_data[0].min := 1.0, [1323].log_data[0].max := 1.0, [1323].log_data[0].total := 300.0, [1323].log_data[0].time := 300.0, [1323].log_data[0].minminute := 45, [1323].log_data[0].maxminute := 45, [1323].log_data[0].valid := 1, [1323].log_data[1].valid := 1, [1323].log_data[2].valid := 1, [1323].log_data[3].valid := 1, [1323].log_data[4].valid := 1, [1323].time.Year := 2022, [1323].time.Month := 4, [1323].time.Day := 28, [1323].time.Hour := 11, [1323].time.Minute := 49, [1323].time.Second := 59, [1323].time.DST_ON := 1, [1324].log_data[0].min := 1.0, [1324].log_data[0].max := 1.0, [1324].log_data[0].total := 300.0, [1324].log_data[0].time := 300.0, [1324].log_data[0].minminute := 50, [1324].log_data[0].maxminute := 50, [1324].log_data[0].valid := 1, [1324].log_data[1].valid := 1, [1324].log_data[2].valid := 1, [1324].log_data[3].valid := 1, [1324].log_data[4].valid := 1, [1324].time.Year := 2022, [1324].time.Month := 4, [1324].time.Day := 28, [1324].time.Hour := 11, [1324].time.Minute := 54, [1324].time.Second := 59, [1324].time.DST_ON := 1, [1325].log_data[0].min := 1.0, [1325].log_data[0].max := 1.0, [1325].log_data[0].total := 300.0, [1325].log_data[0].time := 300.0, [1325].log_data[0].minminute := 55,
        [1325].log_data[0].maxminute := 55, [1325].log_data[0].valid := 1, [1325].log_data[1].valid := 1, [1325].log_data[2].valid := 1, [1325].log_data[3].valid := 1, [1325].log_data[4].valid := 1, [1325].time.Year := 2022, [1325].time.Month := 4, [1325].time.Day := 28, [1325].time.Hour := 11, [1325].time.Minute := 59, [1325].time.Second := 59, [1325].time.DST_ON := 1, [1326].log_data[0].min := 1.0, [1326].log_data[0].max := 1.0, [1326].log_data[0].total := 300.0, [1326].log_data[0].time := 300.0, [1326].log_data[0].valid := 1, [1326].log_data[1].valid := 1, [1326].log_data[2].valid := 1, [1326].log_data[3].valid := 1, [1326].log_data[4].valid := 1, [1326].time.Year := 2022, [1326].time.Month := 4, [1326].time.Day := 28, [1326].time.Hour := 12, [1326].time.Minute := 4, [1326].time.Second := 59, [1326].time.DST_ON := 1, [1327].log_data[0].min := 1.0, [1327].log_data[0].max := 1.0, [1327].log_data[0].total := 300.0, [1327].log_data[0].time := 300.0, [1327].log_data[0].minminute := 5, [1327].log_data[0].maxminute := 5, [1327].log_data[0].valid := 1, [1327].log_data[1].valid := 1, [1327].log_data[2].valid := 1, [1327].log_data[3].valid := 1, [1327].log_data[4].valid := 1, [1327].time.Year := 2022, [1327].time.Month := 4, [1327].time.Day := 28, [1327].time.Hour := 12, [1327].time.Minute := 9, [1327].time.Second := 59, [1327].time.DST_ON := 1, [1328].log_data[0].min := 1.0, [1328].log_data[0].max := 1.0, [1328].log_data[0].total := 300.0, [1328].log_data[0].time := 300.0, [1328].log_data[0].minminute := 10, [1328].log_data[0].maxminute := 10, [1328].log_data[0].valid := 1, [1328].log_data[1].valid := 1, [1328].log_data[2].valid := 1, [1328].log_data[3].valid := 1, [1328].log_data[4].valid := 1, [1328].time.Year := 2022, [1328].time.Month := 4,
        [1328].time.Day := 28, [1328].time.Hour := 12, [1328].time.Minute := 14, [1328].time.Second := 59, [1328].time.DST_ON := 1, [1329].log_data[0].min := 1.0, [1329].log_data[0].max := 1.0, [1329].log_data[0].total := 300.0, [1329].log_data[0].time := 300.0, [1329].log_data[0].minminute := 15, [1329].log_data[0].maxminute := 15, [1329].log_data[0].valid := 1, [1329].log_data[1].valid := 1, [1329].log_data[2].valid := 1, [1329].log_data[3].valid := 1, [1329].log_data[4].valid := 1, [1329].time.Year := 2022, [1329].time.Month := 4, [1329].time.Day := 28, [1329].time.Hour := 12, [1329].time.Minute := 19, [1329].time.Second := 59, [1329].time.DST_ON := 1, [1330].log_data[0].min := 1.0, [1330].log_data[0].max := 1.0, [1330].log_data[0].total := 300.0, [1330].log_data[0].time := 300.0, [1330].log_data[0].minminute := 20, [1330].log_data[0].maxminute := 20, [1330].log_data[0].valid := 1, [1330].log_data[1].valid := 1, [1330].log_data[2].valid := 1, [1330].log_data[3].valid := 1, [1330].log_data[4].valid := 1, [1330].time.Year := 2022, [1330].time.Month := 4, [1330].time.Day := 28, [1330].time.Hour := 12, [1330].time.Minute := 24, [1330].time.Second := 59, [1330].time.DST_ON := 1, [1331].log_data[0].min := 1.0, [1331].log_data[0].max := 1.0, [1331].log_data[0].total := 300.0, [1331].log_data[0].time := 300.0, [1331].log_data[0].minminute := 25, [1331].log_data[0].maxminute := 25, [1331].log_data[0].valid := 1, [1331].log_data[1].valid := 1, [1331].log_data[2].valid := 1, [1331].log_data[3].valid := 1, [1331].log_data[4].valid := 1, [1331].time.Year := 2022, [1331].time.Month := 4, [1331].time.Day := 28, [1331].time.Hour := 12, [1331].time.Minute := 29, [1331].time.Second := 59, [1331].time.DST_ON := 1, [1332].log_data[0].min := 1.0,
        [1332].log_data[0].max := 1.0, [1332].log_data[0].total := 300.0, [1332].log_data[0].time := 300.0, [1332].log_data[0].minminute := 30, [1332].log_data[0].maxminute := 30, [1332].log_data[0].valid := 1, [1332].log_data[1].valid := 1, [1332].log_data[2].valid := 1, [1332].log_data[3].valid := 1, [1332].log_data[4].valid := 1, [1332].time.Year := 2022, [1332].time.Month := 4, [1332].time.Day := 28, [1332].time.Hour := 12, [1332].time.Minute := 34, [1332].time.Second := 59, [1332].time.DST_ON := 1, [1333].log_data[0].min := 1.0, [1333].log_data[0].max := 1.0, [1333].log_data[0].total := 300.0, [1333].log_data[0].time := 300.0, [1333].log_data[0].minminute := 35, [1333].log_data[0].maxminute := 35, [1333].log_data[0].valid := 1, [1333].log_data[1].valid := 1, [1333].log_data[2].valid := 1, [1333].log_data[3].valid := 1, [1333].log_data[4].valid := 1, [1333].time.Year := 2022, [1333].time.Month := 4, [1333].time.Day := 28, [1333].time.Hour := 12, [1333].time.Minute := 39, [1333].time.Second := 59, [1333].time.DST_ON := 1, [1334].log_data[0].min := 1.0, [1334].log_data[0].max := 1.0, [1334].log_data[0].total := 300.0, [1334].log_data[0].time := 300.0, [1334].log_data[0].minminute := 40, [1334].log_data[0].maxminute := 40, [1334].log_data[0].valid := 1, [1334].log_data[1].valid := 1, [1334].log_data[2].valid := 1, [1334].log_data[3].valid := 1, [1334].log_data[4].valid := 1, [1334].time.Year := 2022, [1334].time.Month := 4, [1334].time.Day := 28, [1334].time.Hour := 12, [1334].time.Minute := 44, [1334].time.Second := 59, [1334].time.DST_ON := 1, [1335].log_data[0].min := 1.0, [1335].log_data[0].max := 1.0, [1335].log_data[0].total := 300.0, [1335].log_data[0].time := 300.0, [1335].log_data[0].minminute := 45, [1335].log_data[0].maxminute := 45, [1335].log_data[0].valid := 1,
        [1335].log_data[1].valid := 1, [1335].log_data[2].valid := 1, [1335].log_data[3].valid := 1, [1335].log_data[4].valid := 1, [1335].time.Year := 2022, [1335].time.Month := 4, [1335].time.Day := 28, [1335].time.Hour := 12, [1335].time.Minute := 49, [1335].time.Second := 59, [1335].time.DST_ON := 1, [1336].log_data[0].min := 1.0, [1336].log_data[0].max := 1.0, [1336].log_data[0].total := 300.0, [1336].log_data[0].time := 300.0, [1336].log_data[0].minminute := 50, [1336].log_data[0].maxminute := 50, [1336].log_data[0].valid := 1, [1336].log_data[1].valid := 1, [1336].log_data[2].valid := 1, [1336].log_data[3].valid := 1, [1336].log_data[4].valid := 1, [1336].time.Year := 2022, [1336].time.Month := 4, [1336].time.Day := 28, [1336].time.Hour := 12, [1336].time.Minute := 54, [1336].time.Second := 59, [1336].time.DST_ON := 1, [1337].log_data[0].min := 1.0, [1337].log_data[0].max := 1.0, [1337].log_data[0].total := 300.0, [1337].log_data[0].time := 300.0, [1337].log_data[0].minminute := 55, [1337].log_data[0].maxminute := 55, [1337].log_data[0].valid := 1, [1337].log_data[1].valid := 1, [1337].log_data[2].valid := 1, [1337].log_data[3].valid := 1, [1337].log_data[4].valid := 1, [1337].time.Year := 2022, [1337].time.Month := 4, [1337].time.Day := 28, [1337].time.Hour := 12, [1337].time.Minute := 59, [1337].time.Second := 59, [1337].time.DST_ON := 1, [1338].log_data[0].min := 1.0, [1338].log_data[0].max := 1.0, [1338].log_data[0].total := 300.0, [1338].log_data[0].time := 300.0, [1338].log_data[0].valid := 1, [1338].log_data[1].valid := 1, [1338].log_data[2].valid := 1, [1338].log_data[3].valid := 1, [1338].log_data[4].valid := 1, [1338].time.Year := 2022, [1338].time.Month := 4, [1338].time.Day := 28, [1338].time.Hour := 13,
        [1338].time.Minute := 4, [1338].time.Second := 59, [1338].time.DST_ON := 1, [1339].log_data[0].min := 1.0, [1339].log_data[0].max := 1.0, [1339].log_data[0].total := 300.0, [1339].log_data[0].time := 300.0, [1339].log_data[0].minminute := 5, [1339].log_data[0].maxminute := 5, [1339].log_data[0].valid := 1, [1339].log_data[1].valid := 1, [1339].log_data[2].valid := 1, [1339].log_data[3].valid := 1, [1339].log_data[4].valid := 1, [1339].time.Year := 2022, [1339].time.Month := 4, [1339].time.Day := 28, [1339].time.Hour := 13, [1339].time.Minute := 9, [1339].time.Second := 59, [1339].time.DST_ON := 1, [1340].log_data[0].min := 1.0, [1340].log_data[0].max := 1.0, [1340].log_data[0].total := 300.0, [1340].log_data[0].time := 300.0, [1340].log_data[0].minminute := 10, [1340].log_data[0].maxminute := 10, [1340].log_data[0].valid := 1, [1340].log_data[1].valid := 1, [1340].log_data[2].valid := 1, [1340].log_data[3].valid := 1, [1340].log_data[4].valid := 1, [1340].time.Year := 2022, [1340].time.Month := 4, [1340].time.Day := 28, [1340].time.Hour := 13, [1340].time.Minute := 14, [1340].time.Second := 59, [1340].time.DST_ON := 1, [1341].log_data[0].min := 1.0, [1341].log_data[0].max := 1.0, [1341].log_data[0].total := 300.0, [1341].log_data[0].time := 300.0, [1341].log_data[0].minminute := 15, [1341].log_data[0].maxminute := 15, [1341].log_data[0].valid := 1, [1341].log_data[1].valid := 1, [1341].log_data[2].valid := 1, [1341].log_data[3].valid := 1, [1341].log_data[4].valid := 1, [1341].time.Year := 2022, [1341].time.Month := 4, [1341].time.Day := 28, [1341].time.Hour := 13, [1341].time.Minute := 19, [1341].time.Second := 59, [1341].time.DST_ON := 1, [1342].log_data[0].min := 1.0, [1342].log_data[0].max := 1.0, [1342].log_data[0].total := 300.0,
        [1342].log_data[0].time := 300.0, [1342].log_data[0].minminute := 20, [1342].log_data[0].maxminute := 20, [1342].log_data[0].valid := 1, [1342].log_data[1].valid := 1, [1342].log_data[2].valid := 1, [1342].log_data[3].valid := 1, [1342].log_data[4].valid := 1, [1342].time.Year := 2022, [1342].time.Month := 4, [1342].time.Day := 28, [1342].time.Hour := 13, [1342].time.Minute := 24, [1342].time.Second := 59, [1342].time.DST_ON := 1, [1343].log_data[0].min := 1.0, [1343].log_data[0].max := 1.0, [1343].log_data[0].total := 300.0, [1343].log_data[0].time := 300.0, [1343].log_data[0].minminute := 25, [1343].log_data[0].maxminute := 25, [1343].log_data[0].valid := 1, [1343].log_data[1].valid := 1, [1343].log_data[2].valid := 1, [1343].log_data[3].valid := 1, [1343].log_data[4].valid := 1, [1343].time.Year := 2022, [1343].time.Month := 4, [1343].time.Day := 28, [1343].time.Hour := 13, [1343].time.Minute := 29, [1343].time.Second := 59, [1343].time.DST_ON := 1, [1344].log_data[0].min := 1.0, [1344].log_data[0].max := 1.0, [1344].log_data[0].total := 300.0, [1344].log_data[0].time := 300.0, [1344].log_data[0].minminute := 30, [1344].log_data[0].maxminute := 30, [1344].log_data[0].valid := 1, [1344].log_data[1].valid := 1, [1344].log_data[2].valid := 1, [1344].log_data[3].valid := 1, [1344].log_data[4].valid := 1, [1344].time.Year := 2022, [1344].time.Month := 4, [1344].time.Day := 28, [1344].time.Hour := 13, [1344].time.Minute := 34, [1344].time.Second := 59, [1344].time.DST_ON := 1, [1345].log_data[0].min := 1.0, [1345].log_data[0].max := 1.0, [1345].log_data[0].total := 300.0, [1345].log_data[0].time := 300.0, [1345].log_data[0].minminute := 35, [1345].log_data[0].maxminute := 35, [1345].log_data[0].valid := 1, [1345].log_data[1].valid := 1, [1345].log_data[2].valid := 1,
        [1345].log_data[3].valid := 1, [1345].log_data[4].valid := 1, [1345].time.Year := 2022, [1345].time.Month := 4, [1345].time.Day := 28, [1345].time.Hour := 13, [1345].time.Minute := 39, [1345].time.Second := 59, [1345].time.DST_ON := 1, [1346].log_data[0].min := 1.0, [1346].log_data[0].max := 1.0, [1346].log_data[0].total := 300.0, [1346].log_data[0].time := 300.0, [1346].log_data[0].minminute := 40, [1346].log_data[0].maxminute := 40, [1346].log_data[0].valid := 1, [1346].log_data[1].valid := 1, [1346].log_data[2].valid := 1, [1346].log_data[3].valid := 1, [1346].log_data[4].valid := 1, [1346].time.Year := 2022, [1346].time.Month := 4, [1346].time.Day := 28, [1346].time.Hour := 13, [1346].time.Minute := 44, [1346].time.Second := 59, [1346].time.DST_ON := 1, [1347].log_data[0].min := 1.0, [1347].log_data[0].max := 1.0, [1347].log_data[0].total := 300.0, [1347].log_data[0].time := 300.0, [1347].log_data[0].minminute := 45, [1347].log_data[0].maxminute := 45, [1347].log_data[0].valid := 1, [1347].log_data[1].valid := 1, [1347].log_data[2].valid := 1, [1347].log_data[3].valid := 1, [1347].log_data[4].valid := 1, [1347].time.Year := 2022, [1347].time.Month := 4, [1347].time.Day := 28, [1347].time.Hour := 13, [1347].time.Minute := 49, [1347].time.Second := 59, [1347].time.DST_ON := 1, [1348].log_data[0].min := 1.0, [1348].log_data[0].max := 1.0, [1348].log_data[0].total := 300.0, [1348].log_data[0].time := 300.0, [1348].log_data[0].minminute := 50, [1348].log_data[0].maxminute := 50, [1348].log_data[0].valid := 1, [1348].log_data[1].valid := 1, [1348].log_data[2].valid := 1, [1348].log_data[3].valid := 1, [1348].log_data[4].valid := 1, [1348].time.Year := 2022, [1348].time.Month := 4, [1348].time.Day := 28, [1348].time.Hour := 13,
        [1348].time.Minute := 54, [1348].time.Second := 59, [1348].time.DST_ON := 1, [1349].log_data[0].min := 1.0, [1349].log_data[0].max := 1.0, [1349].log_data[0].total := 300.0, [1349].log_data[0].time := 300.0, [1349].log_data[0].minminute := 55, [1349].log_data[0].maxminute := 55, [1349].log_data[0].valid := 1, [1349].log_data[1].valid := 1, [1349].log_data[2].valid := 1, [1349].log_data[3].valid := 1, [1349].log_data[4].valid := 1, [1349].time.Year := 2022, [1349].time.Month := 4, [1349].time.Day := 28, [1349].time.Hour := 13, [1349].time.Minute := 59, [1349].time.Second := 59, [1349].time.DST_ON := 1, [1350].log_data[0].min := 1.0, [1350].log_data[0].max := 1.0, [1350].log_data[0].total := 300.0, [1350].log_data[0].time := 300.0, [1350].log_data[0].valid := 1, [1350].log_data[1].valid := 1, [1350].log_data[2].valid := 1, [1350].log_data[3].valid := 1, [1350].log_data[4].valid := 1, [1350].time.Year := 2022, [1350].time.Month := 4, [1350].time.Day := 28, [1350].time.Hour := 14, [1350].time.Minute := 4, [1350].time.Second := 59, [1350].time.DST_ON := 1, [1351].log_data[0].min := 1.0, [1351].log_data[0].max := 1.0, [1351].log_data[0].total := 300.0, [1351].log_data[0].time := 300.0, [1351].log_data[0].minminute := 5, [1351].log_data[0].maxminute := 5, [1351].log_data[0].valid := 1, [1351].log_data[1].valid := 1, [1351].log_data[2].valid := 1, [1351].log_data[3].valid := 1, [1351].log_data[4].valid := 1, [1351].time.Year := 2022, [1351].time.Month := 4, [1351].time.Day := 28, [1351].time.Hour := 14, [1351].time.Minute := 9, [1351].time.Second := 59, [1351].time.DST_ON := 1, [1352].log_data[0].min := 1.0, [1352].log_data[0].max := 1.0, [1352].log_data[0].total := 300.0, [1352].log_data[0].time := 300.0, [1352].log_data[0].minminute := 10,
        [1352].log_data[0].maxminute := 10, [1352].log_data[0].valid := 1, [1352].log_data[1].valid := 1, [1352].log_data[2].valid := 1, [1352].log_data[3].valid := 1, [1352].log_data[4].valid := 1, [1352].time.Year := 2022, [1352].time.Month := 4, [1352].time.Day := 28, [1352].time.Hour := 14, [1352].time.Minute := 14, [1352].time.Second := 59, [1352].time.DST_ON := 1, [1353].log_data[0].min := 1.0, [1353].log_data[0].max := 1.0, [1353].log_data[0].total := 300.0, [1353].log_data[0].time := 300.0, [1353].log_data[0].minminute := 15, [1353].log_data[0].maxminute := 15, [1353].log_data[0].valid := 1, [1353].log_data[1].valid := 1, [1353].log_data[2].valid := 1, [1353].log_data[3].valid := 1, [1353].log_data[4].valid := 1, [1353].time.Year := 2022, [1353].time.Month := 4, [1353].time.Day := 28, [1353].time.Hour := 14, [1353].time.Minute := 19, [1353].time.Second := 59, [1353].time.DST_ON := 1, [1354].log_data[0].min := 1.0, [1354].log_data[0].max := 1.0, [1354].log_data[0].total := 300.0, [1354].log_data[0].time := 300.0, [1354].log_data[0].minminute := 20, [1354].log_data[0].maxminute := 20, [1354].log_data[0].valid := 1, [1354].log_data[1].valid := 1, [1354].log_data[2].valid := 1, [1354].log_data[3].valid := 1, [1354].log_data[4].valid := 1, [1354].time.Year := 2022, [1354].time.Month := 4, [1354].time.Day := 28, [1354].time.Hour := 14, [1354].time.Minute := 24, [1354].time.Second := 59, [1354].time.DST_ON := 1, [1355].log_data[0].min := 1.0, [1355].log_data[0].max := 1.0, [1355].log_data[0].total := 300.0, [1355].log_data[0].time := 300.0, [1355].log_data[0].minminute := 25, [1355].log_data[0].maxminute := 25, [1355].log_data[0].valid := 1, [1355].log_data[1].valid := 1, [1355].log_data[2].valid := 1, [1355].log_data[3].valid := 1, [1355].log_data[4].valid := 1,
        [1355].time.Year := 2022, [1355].time.Month := 4, [1355].time.Day := 28, [1355].time.Hour := 14, [1355].time.Minute := 29, [1355].time.Second := 59, [1355].time.DST_ON := 1, [1356].log_data[0].min := 1.0, [1356].log_data[0].max := 1.0, [1356].log_data[0].total := 300.0, [1356].log_data[0].time := 300.0, [1356].log_data[0].minminute := 30, [1356].log_data[0].maxminute := 30, [1356].log_data[0].valid := 1, [1356].log_data[1].valid := 1, [1356].log_data[2].valid := 1, [1356].log_data[3].valid := 1, [1356].log_data[4].valid := 1, [1356].time.Year := 2022, [1356].time.Month := 4, [1356].time.Day := 28, [1356].time.Hour := 14, [1356].time.Minute := 34, [1356].time.Second := 59, [1356].time.DST_ON := 1, [1357].log_data[0].min := 1.0, [1357].log_data[0].max := 1.0, [1357].log_data[0].total := 300.0, [1357].log_data[0].time := 300.0, [1357].log_data[0].minminute := 35, [1357].log_data[0].maxminute := 35, [1357].log_data[0].valid := 1, [1357].log_data[1].valid := 1, [1357].log_data[2].valid := 1, [1357].log_data[3].valid := 1, [1357].log_data[4].valid := 1, [1357].time.Year := 2022, [1357].time.Month := 4, [1357].time.Day := 28, [1357].time.Hour := 14, [1357].time.Minute := 39, [1357].time.Second := 59, [1357].time.DST_ON := 1, [1358].log_data[0].min := 1.0, [1358].log_data[0].max := 1.0, [1358].log_data[0].total := 300.0, [1358].log_data[0].time := 300.0, [1358].log_data[0].minminute := 40, [1358].log_data[0].maxminute := 40, [1358].log_data[0].valid := 1, [1358].log_data[1].valid := 1, [1358].log_data[2].valid := 1, [1358].log_data[3].valid := 1, [1358].log_data[4].valid := 1, [1358].time.Year := 2022, [1358].time.Month := 4, [1358].time.Day := 28, [1358].time.Hour := 14, [1358].time.Minute := 44, [1358].time.Second := 59,
        [1358].time.DST_ON := 1, [1359].log_data[0].min := 1.0, [1359].log_data[0].max := 1.0, [1359].log_data[0].total := 300.0, [1359].log_data[0].time := 300.0, [1359].log_data[0].minminute := 45, [1359].log_data[0].maxminute := 45, [1359].log_data[0].valid := 1, [1359].log_data[1].valid := 1, [1359].log_data[2].valid := 1, [1359].log_data[3].valid := 1, [1359].log_data[4].valid := 1, [1359].time.Year := 2022, [1359].time.Month := 4, [1359].time.Day := 28, [1359].time.Hour := 14, [1359].time.Minute := 49, [1359].time.Second := 59, [1359].time.DST_ON := 1, [1360].log_data[0].min := 1.0, [1360].log_data[0].max := 1.0, [1360].log_data[0].total := 300.0, [1360].log_data[0].time := 300.0, [1360].log_data[0].minminute := 50, [1360].log_data[0].maxminute := 50, [1360].log_data[0].valid := 1, [1360].log_data[1].valid := 1, [1360].log_data[2].valid := 1, [1360].log_data[3].valid := 1, [1360].log_data[4].valid := 1, [1360].time.Year := 2022, [1360].time.Month := 4, [1360].time.Day := 28, [1360].time.Hour := 14, [1360].time.Minute := 54, [1360].time.Second := 59, [1360].time.DST_ON := 1, [1361].log_data[0].min := 1.0, [1361].log_data[0].max := 1.0, [1361].log_data[0].total := 299.999, [1361].log_data[0].time := 299.999, [1361].log_data[0].minminute := 55, [1361].log_data[0].maxminute := 55, [1361].log_data[0].valid := 1, [1361].log_data[1].valid := 1, [1361].log_data[2].valid := 1, [1361].log_data[3].valid := 1, [1361].log_data[4].valid := 1, [1361].time.Year := 2022, [1361].time.Month := 4, [1361].time.Day := 28, [1361].time.Hour := 14, [1361].time.Minute := 59, [1361].time.Second := 59, [1361].time.DST_ON := 1, [1362].log_data[0].min := 1.0, [1362].log_data[0].max := 1.0, [1362].log_data[0].total := 300.0, [1362].log_data[0].time := 300.0, [1362].log_data[0].valid := 1,
        [1362].log_data[1].valid := 1, [1362].log_data[2].valid := 1, [1362].log_data[3].valid := 1, [1362].log_data[4].valid := 1, [1362].time.Year := 2022, [1362].time.Month := 4, [1362].time.Day := 28, [1362].time.Hour := 15, [1362].time.Minute := 4, [1362].time.Second := 59, [1362].time.DST_ON := 1, [1363].log_data[0].min := 1.0, [1363].log_data[0].max := 1.0, [1363].log_data[0].total := 300.0, [1363].log_data[0].time := 300.0, [1363].log_data[0].minminute := 5, [1363].log_data[0].maxminute := 5, [1363].log_data[0].valid := 1, [1363].log_data[1].valid := 1, [1363].log_data[2].valid := 1, [1363].log_data[3].valid := 1, [1363].log_data[4].valid := 1, [1363].time.Year := 2022, [1363].time.Month := 4, [1363].time.Day := 28, [1363].time.Hour := 15, [1363].time.Minute := 9, [1363].time.Second := 59, [1363].time.DST_ON := 1, [1364].log_data[0].min := 1.0, [1364].log_data[0].max := 1.0, [1364].log_data[0].total := 300.0, [1364].log_data[0].time := 300.0, [1364].log_data[0].minminute := 10, [1364].log_data[0].maxminute := 10, [1364].log_data[0].valid := 1, [1364].log_data[1].valid := 1, [1364].log_data[2].valid := 1, [1364].log_data[3].valid := 1, [1364].log_data[4].valid := 1, [1364].time.Year := 2022, [1364].time.Month := 4, [1364].time.Day := 28, [1364].time.Hour := 15, [1364].time.Minute := 14, [1364].time.Second := 59, [1364].time.DST_ON := 1, [1365].log_data[0].min := 1.0, [1365].log_data[0].max := 1.0, [1365].log_data[0].total := 300.0, [1365].log_data[0].time := 300.0, [1365].log_data[0].minminute := 15, [1365].log_data[0].maxminute := 15, [1365].log_data[0].valid := 1, [1365].log_data[1].valid := 1, [1365].log_data[2].valid := 1, [1365].log_data[3].valid := 1, [1365].log_data[4].valid := 1, [1365].time.Year := 2022, [1365].time.Month := 4,
        [1365].time.Day := 28, [1365].time.Hour := 15, [1365].time.Minute := 19, [1365].time.Second := 59, [1365].time.DST_ON := 1, [1366].log_data[0].min := 1.0, [1366].log_data[0].max := 1.0, [1366].log_data[0].total := 300.0, [1366].log_data[0].time := 300.0, [1366].log_data[0].minminute := 20, [1366].log_data[0].maxminute := 20, [1366].log_data[0].valid := 1, [1366].log_data[1].valid := 1, [1366].log_data[2].valid := 1, [1366].log_data[3].valid := 1, [1366].log_data[4].valid := 1, [1366].time.Year := 2022, [1366].time.Month := 4, [1366].time.Day := 28, [1366].time.Hour := 15, [1366].time.Minute := 24, [1366].time.Second := 59, [1366].time.DST_ON := 1, [1367].log_data[0].min := 1.0, [1367].log_data[0].max := 1.0, [1367].log_data[0].total := 300.0, [1367].log_data[0].time := 300.0, [1367].log_data[0].minminute := 25, [1367].log_data[0].maxminute := 25, [1367].log_data[0].valid := 1, [1367].log_data[1].valid := 1, [1367].log_data[2].valid := 1, [1367].log_data[3].valid := 1, [1367].log_data[4].valid := 1, [1367].time.Year := 2022, [1367].time.Month := 4, [1367].time.Day := 28, [1367].time.Hour := 15, [1367].time.Minute := 29, [1367].time.Second := 59, [1367].time.DST_ON := 1, [1368].log_data[0].min := 1.0, [1368].log_data[0].max := 1.0, [1368].log_data[0].total := 300.0, [1368].log_data[0].time := 300.0, [1368].log_data[0].minminute := 30, [1368].log_data[0].maxminute := 30, [1368].log_data[0].valid := 1, [1368].log_data[1].valid := 1, [1368].log_data[2].valid := 1, [1368].log_data[3].valid := 1, [1368].log_data[4].valid := 1, [1368].time.Year := 2022, [1368].time.Month := 4, [1368].time.Day := 28, [1368].time.Hour := 15, [1368].time.Minute := 34, [1368].time.Second := 59, [1368].time.DST_ON := 1, [1369].log_data[0].min := 1.0,
        [1369].log_data[0].max := 1.0, [1369].log_data[0].total := 300.0, [1369].log_data[0].time := 300.0, [1369].log_data[0].minminute := 35, [1369].log_data[0].maxminute := 35, [1369].log_data[0].valid := 1, [1369].log_data[1].valid := 1, [1369].log_data[2].valid := 1, [1369].log_data[3].valid := 1, [1369].log_data[4].valid := 1, [1369].time.Year := 2022, [1369].time.Month := 4, [1369].time.Day := 28, [1369].time.Hour := 15, [1369].time.Minute := 39, [1369].time.Second := 59, [1369].time.DST_ON := 1, [1370].log_data[0].min := 1.0, [1370].log_data[0].max := 1.0, [1370].log_data[0].total := 300.0, [1370].log_data[0].time := 300.0, [1370].log_data[0].minminute := 40, [1370].log_data[0].maxminute := 40, [1370].log_data[0].valid := 1, [1370].log_data[1].valid := 1, [1370].log_data[2].valid := 1, [1370].log_data[3].valid := 1, [1370].log_data[4].valid := 1, [1370].time.Year := 2022, [1370].time.Month := 4, [1370].time.Day := 28, [1370].time.Hour := 15, [1370].time.Minute := 44, [1370].time.Second := 59, [1370].time.DST_ON := 1, [1371].log_data[0].min := 1.0, [1371].log_data[0].max := 1.0, [1371].log_data[0].total := 300.0, [1371].log_data[0].time := 300.0, [1371].log_data[0].minminute := 45, [1371].log_data[0].maxminute := 45, [1371].log_data[0].valid := 1, [1371].log_data[1].valid := 1, [1371].log_data[2].valid := 1, [1371].log_data[3].valid := 1, [1371].log_data[4].valid := 1, [1371].time.Year := 2022, [1371].time.Month := 4, [1371].time.Day := 28, [1371].time.Hour := 15, [1371].time.Minute := 49, [1371].time.Second := 59, [1371].time.DST_ON := 1, [1372].log_data[0].min := 1.0, [1372].log_data[0].max := 1.0, [1372].log_data[0].total := 300.0, [1372].log_data[0].time := 300.0, [1372].log_data[0].minminute := 50, [1372].log_data[0].maxminute := 50, [1372].log_data[0].valid := 1,
        [1372].log_data[1].valid := 1, [1372].log_data[2].valid := 1, [1372].log_data[3].valid := 1, [1372].log_data[4].valid := 1, [1372].time.Year := 2022, [1372].time.Month := 4, [1372].time.Day := 28, [1372].time.Hour := 15, [1372].time.Minute := 54, [1372].time.Second := 59, [1372].time.DST_ON := 1, [1373].log_data[0].min := 1.0, [1373].log_data[0].max := 1.0, [1373].log_data[0].total := 300.0, [1373].log_data[0].time := 300.0, [1373].log_data[0].minminute := 55, [1373].log_data[0].maxminute := 55, [1373].log_data[0].valid := 1, [1373].log_data[1].valid := 1, [1373].log_data[2].valid := 1, [1373].log_data[3].valid := 1, [1373].log_data[4].valid := 1, [1373].time.Year := 2022, [1373].time.Month := 4, [1373].time.Day := 28, [1373].time.Hour := 15, [1373].time.Minute := 59, [1373].time.Second := 59, [1373].time.DST_ON := 1, [1374].log_data[0].min := 1.0, [1374].log_data[0].max := 1.0, [1374].log_data[0].total := 300.0, [1374].log_data[0].time := 300.0, [1374].log_data[0].valid := 1, [1374].log_data[1].valid := 1, [1374].log_data[2].valid := 1, [1374].log_data[3].valid := 1, [1374].log_data[4].valid := 1, [1374].time.Year := 2022, [1374].time.Month := 4, [1374].time.Day := 28, [1374].time.Hour := 16, [1374].time.Minute := 4, [1374].time.Second := 59, [1374].time.DST_ON := 1, [1375].log_data[0].min := 1.0, [1375].log_data[0].max := 1.0, [1375].log_data[0].total := 300.0, [1375].log_data[0].time := 300.0, [1375].log_data[0].minminute := 5, [1375].log_data[0].maxminute := 5, [1375].log_data[0].valid := 1, [1375].log_data[1].valid := 1, [1375].log_data[2].valid := 1, [1375].log_data[3].valid := 1, [1375].log_data[4].valid := 1, [1375].time.Year := 2022, [1375].time.Month := 4, [1375].time.Day := 28, [1375].time.Hour := 16,
        [1375].time.Minute := 9, [1375].time.Second := 59, [1375].time.DST_ON := 1, [1376].log_data[0].min := 1.0, [1376].log_data[0].max := 1.0, [1376].log_data[0].total := 300.0, [1376].log_data[0].time := 300.0, [1376].log_data[0].minminute := 10, [1376].log_data[0].maxminute := 10, [1376].log_data[0].valid := 1, [1376].log_data[1].valid := 1, [1376].log_data[2].valid := 1, [1376].log_data[3].valid := 1, [1376].log_data[4].valid := 1, [1376].time.Year := 2022, [1376].time.Month := 4, [1376].time.Day := 28, [1376].time.Hour := 16, [1376].time.Minute := 14, [1376].time.Second := 59, [1376].time.DST_ON := 1, [1377].log_data[0].min := 1.0, [1377].log_data[0].max := 1.0, [1377].log_data[0].total := 300.0, [1377].log_data[0].time := 300.0, [1377].log_data[0].minminute := 15, [1377].log_data[0].maxminute := 15, [1377].log_data[0].valid := 1, [1377].log_data[1].valid := 1, [1377].log_data[2].valid := 1, [1377].log_data[3].valid := 1, [1377].log_data[4].valid := 1, [1377].time.Year := 2022, [1377].time.Month := 4, [1377].time.Day := 28, [1377].time.Hour := 16, [1377].time.Minute := 19, [1377].time.Second := 59, [1377].time.DST_ON := 1, [1378].log_data[0].min := 1.0, [1378].log_data[0].max := 1.0, [1378].log_data[0].total := 300.0, [1378].log_data[0].time := 300.0, [1378].log_data[0].minminute := 20, [1378].log_data[0].maxminute := 20, [1378].log_data[0].valid := 1, [1378].log_data[1].valid := 1, [1378].log_data[2].valid := 1, [1378].log_data[3].valid := 1, [1378].log_data[4].valid := 1, [1378].time.Year := 2022, [1378].time.Month := 4, [1378].time.Day := 28, [1378].time.Hour := 16, [1378].time.Minute := 24, [1378].time.Second := 59, [1378].time.DST_ON := 1, [1379].log_data[0].min := 1.0, [1379].log_data[0].max := 1.0, [1379].log_data[0].total := 300.0,
        [1379].log_data[0].time := 300.0, [1379].log_data[0].minminute := 25, [1379].log_data[0].maxminute := 25, [1379].log_data[0].valid := 1, [1379].log_data[1].valid := 1, [1379].log_data[2].valid := 1, [1379].log_data[3].valid := 1, [1379].log_data[4].valid := 1, [1379].time.Year := 2022, [1379].time.Month := 4, [1379].time.Day := 28, [1379].time.Hour := 16, [1379].time.Minute := 29, [1379].time.Second := 59, [1379].time.DST_ON := 1, [1380].log_data[0].min := 1.0, [1380].log_data[0].max := 1.0, [1380].log_data[0].total := 300.0, [1380].log_data[0].time := 300.0, [1380].log_data[0].minminute := 30, [1380].log_data[0].maxminute := 30, [1380].log_data[0].valid := 1, [1380].log_data[1].valid := 1, [1380].log_data[2].valid := 1, [1380].log_data[3].valid := 1, [1380].log_data[4].valid := 1, [1380].time.Year := 2022, [1380].time.Month := 4, [1380].time.Day := 28, [1380].time.Hour := 16, [1380].time.Minute := 34, [1380].time.Second := 59, [1380].time.DST_ON := 1, [1381].log_data[0].min := 1.0, [1381].log_data[0].max := 1.0, [1381].log_data[0].total := 300.0, [1381].log_data[0].time := 300.0, [1381].log_data[0].minminute := 35, [1381].log_data[0].maxminute := 35, [1381].log_data[0].valid := 1, [1381].log_data[1].valid := 1, [1381].log_data[2].valid := 1, [1381].log_data[3].valid := 1, [1381].log_data[4].valid := 1, [1381].time.Year := 2022, [1381].time.Month := 4, [1381].time.Day := 28, [1381].time.Hour := 16, [1381].time.Minute := 39, [1381].time.Second := 59, [1381].time.DST_ON := 1, [1382].log_data[0].min := 1.0, [1382].log_data[0].max := 1.0, [1382].log_data[0].total := 300.0, [1382].log_data[0].time := 300.0, [1382].log_data[0].minminute := 40, [1382].log_data[0].maxminute := 40, [1382].log_data[0].valid := 1, [1382].log_data[1].valid := 1, [1382].log_data[2].valid := 1,
        [1382].log_data[3].valid := 1, [1382].log_data[4].valid := 1, [1382].time.Year := 2022, [1382].time.Month := 4, [1382].time.Day := 28, [1382].time.Hour := 16, [1382].time.Minute := 44, [1382].time.Second := 59, [1382].time.DST_ON := 1, [1383].log_data[0].min := 1.0, [1383].log_data[0].max := 1.0, [1383].log_data[0].total := 300.0, [1383].log_data[0].time := 300.0, [1383].log_data[0].minminute := 45, [1383].log_data[0].maxminute := 45, [1383].log_data[0].valid := 1, [1383].log_data[1].valid := 1, [1383].log_data[2].valid := 1, [1383].log_data[3].valid := 1, [1383].log_data[4].valid := 1, [1383].time.Year := 2022, [1383].time.Month := 4, [1383].time.Day := 28, [1383].time.Hour := 16, [1383].time.Minute := 49, [1383].time.Second := 59, [1383].time.DST_ON := 1, [1384].log_data[0].min := 1.0, [1384].log_data[0].max := 1.0, [1384].log_data[0].total := 300.0, [1384].log_data[0].time := 300.0, [1384].log_data[0].minminute := 50, [1384].log_data[0].maxminute := 50, [1384].log_data[0].valid := 1, [1384].log_data[1].valid := 1, [1384].log_data[2].valid := 1, [1384].log_data[3].valid := 1, [1384].log_data[4].valid := 1, [1384].time.Year := 2022, [1384].time.Month := 4, [1384].time.Day := 28, [1384].time.Hour := 16, [1384].time.Minute := 54, [1384].time.Second := 59, [1384].time.DST_ON := 1, [1385].log_data[0].min := 1.0, [1385].log_data[0].max := 1.0, [1385].log_data[0].total := 300.0, [1385].log_data[0].time := 300.0, [1385].log_data[0].minminute := 55, [1385].log_data[0].maxminute := 55, [1385].log_data[0].valid := 1, [1385].log_data[1].valid := 1, [1385].log_data[2].valid := 1, [1385].log_data[3].valid := 1, [1385].log_data[4].valid := 1, [1385].time.Year := 2022, [1385].time.Month := 4, [1385].time.Day := 28, [1385].time.Hour := 16,
        [1385].time.Minute := 59, [1385].time.Second := 59, [1385].time.DST_ON := 1, [1386].log_data[0].min := 1.0, [1386].log_data[0].max := 1.0, [1386].log_data[0].total := 300.0, [1386].log_data[0].time := 300.0, [1386].log_data[0].valid := 1, [1386].log_data[1].valid := 1, [1386].log_data[2].valid := 1, [1386].log_data[3].valid := 1, [1386].log_data[4].valid := 1, [1386].time.Year := 2022, [1386].time.Month := 4, [1386].time.Day := 28, [1386].time.Hour := 17, [1386].time.Minute := 4, [1386].time.Second := 59, [1386].time.DST_ON := 1, [1387].log_data[0].min := 1.0, [1387].log_data[0].max := 1.0, [1387].log_data[0].total := 300.0, [1387].log_data[0].time := 300.0, [1387].log_data[0].minminute := 5, [1387].log_data[0].maxminute := 5, [1387].log_data[0].valid := 1, [1387].log_data[1].valid := 1, [1387].log_data[2].valid := 1, [1387].log_data[3].valid := 1, [1387].log_data[4].valid := 1, [1387].time.Year := 2022, [1387].time.Month := 4, [1387].time.Day := 28, [1387].time.Hour := 17, [1387].time.Minute := 9, [1387].time.Second := 59, [1387].time.DST_ON := 1, [1388].log_data[0].min := 1.0, [1388].log_data[0].max := 1.0, [1388].log_data[0].total := 300.0, [1388].log_data[0].time := 300.0, [1388].log_data[0].minminute := 10, [1388].log_data[0].maxminute := 10, [1388].log_data[0].valid := 1, [1388].log_data[1].valid := 1, [1388].log_data[2].valid := 1, [1388].log_data[3].valid := 1, [1388].log_data[4].valid := 1, [1388].time.Year := 2022, [1388].time.Month := 4, [1388].time.Day := 28, [1388].time.Hour := 17, [1388].time.Minute := 14, [1388].time.Second := 59, [1388].time.DST_ON := 1, [1389].log_data[0].min := 1.0, [1389].log_data[0].max := 1.0, [1389].log_data[0].total := 300.0, [1389].log_data[0].time := 300.0, [1389].log_data[0].minminute := 15,
        [1389].log_data[0].maxminute := 15, [1389].log_data[0].valid := 1, [1389].log_data[1].valid := 1, [1389].log_data[2].valid := 1, [1389].log_data[3].valid := 1, [1389].log_data[4].valid := 1, [1389].time.Year := 2022, [1389].time.Month := 4, [1389].time.Day := 28, [1389].time.Hour := 17, [1389].time.Minute := 19, [1389].time.Second := 59, [1389].time.DST_ON := 1, [1390].log_data[0].min := 1.0, [1390].log_data[0].max := 1.0, [1390].log_data[0].total := 300.0, [1390].log_data[0].time := 300.0, [1390].log_data[0].minminute := 20, [1390].log_data[0].maxminute := 20, [1390].log_data[0].valid := 1, [1390].log_data[1].valid := 1, [1390].log_data[2].valid := 1, [1390].log_data[3].valid := 1, [1390].log_data[4].valid := 1, [1390].time.Year := 2022, [1390].time.Month := 4, [1390].time.Day := 28, [1390].time.Hour := 17, [1390].time.Minute := 24, [1390].time.Second := 59, [1390].time.DST_ON := 1, [1391].log_data[0].min := 1.0, [1391].log_data[0].max := 1.0, [1391].log_data[0].total := 300.5, [1391].log_data[0].time := 300.5, [1391].log_data[0].minminute := 25, [1391].log_data[0].maxminute := 25, [1391].log_data[0].valid := 1, [1391].log_data[1].valid := 1, [1391].log_data[2].valid := 1, [1391].log_data[3].valid := 1, [1391].log_data[4].valid := 1, [1391].time.Year := 2022, [1391].time.Month := 4, [1391].time.Day := 28, [1391].time.Hour := 17, [1391].time.Minute := 29, [1391].time.Second := 59, [1391].time.DST_ON := 1, [1392].log_data[0].min := 1.0, [1392].log_data[0].max := 1.0, [1392].log_data[0].total := 300.0, [1392].log_data[0].time := 300.0, [1392].log_data[0].minminute := 30, [1392].log_data[0].maxminute := 30, [1392].log_data[0].valid := 1, [1392].log_data[1].valid := 1, [1392].log_data[2].valid := 1, [1392].log_data[3].valid := 1, [1392].log_data[4].valid := 1,
        [1392].time.Year := 2022, [1392].time.Month := 4, [1392].time.Day := 28, [1392].time.Hour := 17, [1392].time.Minute := 34, [1392].time.Second := 59, [1392].time.DST_ON := 1, [1393].log_data[0].min := 1.0, [1393].log_data[0].max := 1.0, [1393].log_data[0].total := 300.0, [1393].log_data[0].time := 300.0, [1393].log_data[0].minminute := 35, [1393].log_data[0].maxminute := 35, [1393].log_data[0].valid := 1, [1393].log_data[1].valid := 1, [1393].log_data[2].valid := 1, [1393].log_data[3].valid := 1, [1393].log_data[4].valid := 1, [1393].time.Year := 2022, [1393].time.Month := 4, [1393].time.Day := 28, [1393].time.Hour := 17, [1393].time.Minute := 39, [1393].time.Second := 59, [1393].time.DST_ON := 1, [1394].log_data[0].min := 1.0, [1394].log_data[0].max := 1.0, [1394].log_data[0].total := 300.0, [1394].log_data[0].time := 300.0, [1394].log_data[0].minminute := 40, [1394].log_data[0].maxminute := 40, [1394].log_data[0].valid := 1, [1394].log_data[1].valid := 1, [1394].log_data[2].valid := 1, [1394].log_data[3].valid := 1, [1394].log_data[4].valid := 1, [1394].time.Year := 2022, [1394].time.Month := 4, [1394].time.Day := 28, [1394].time.Hour := 17, [1394].time.Minute := 44, [1394].time.Second := 59, [1394].time.DST_ON := 1, [1395].log_data[0].min := 1.0, [1395].log_data[0].max := 1.0, [1395].log_data[0].total := 300.0, [1395].log_data[0].time := 300.0, [1395].log_data[0].minminute := 45, [1395].log_data[0].maxminute := 45, [1395].log_data[0].valid := 1, [1395].log_data[1].valid := 1, [1395].log_data[2].valid := 1, [1395].log_data[3].valid := 1, [1395].log_data[4].valid := 1, [1395].time.Year := 2022, [1395].time.Month := 4, [1395].time.Day := 28, [1395].time.Hour := 17, [1395].time.Minute := 49, [1395].time.Second := 59,
        [1395].time.DST_ON := 1, [1396].log_data[0].min := 1.0, [1396].log_data[0].max := 1.0, [1396].log_data[0].total := 300.0, [1396].log_data[0].time := 300.0, [1396].log_data[0].minminute := 50, [1396].log_data[0].maxminute := 50, [1396].log_data[0].valid := 1, [1396].log_data[1].valid := 1, [1396].log_data[2].valid := 1, [1396].log_data[3].valid := 1, [1396].log_data[4].valid := 1, [1396].time.Year := 2022, [1396].time.Month := 4, [1396].time.Day := 28, [1396].time.Hour := 17, [1396].time.Minute := 54, [1396].time.Second := 59, [1396].time.DST_ON := 1, [1397].log_data[0].min := 1.0, [1397].log_data[0].max := 1.0, [1397].log_data[0].total := 300.0, [1397].log_data[0].time := 300.0, [1397].log_data[0].minminute := 55, [1397].log_data[0].maxminute := 55, [1397].log_data[0].valid := 1, [1397].log_data[1].valid := 1, [1397].log_data[2].valid := 1, [1397].log_data[3].valid := 1, [1397].log_data[4].valid := 1, [1397].time.Year := 2022, [1397].time.Month := 4, [1397].time.Day := 28, [1397].time.Hour := 17, [1397].time.Minute := 59, [1397].time.Second := 59, [1397].time.DST_ON := 1, [1398].log_data[0].min := 1.0, [1398].log_data[0].max := 1.0, [1398].log_data[0].total := 300.0, [1398].log_data[0].time := 300.0, [1398].log_data[0].valid := 1, [1398].log_data[1].valid := 1, [1398].log_data[2].valid := 1, [1398].log_data[3].valid := 1, [1398].log_data[4].valid := 1, [1398].time.Year := 2022, [1398].time.Month := 4, [1398].time.Day := 28, [1398].time.Hour := 18, [1398].time.Minute := 4, [1398].time.Second := 59, [1398].time.DST_ON := 1, [1399].log_data[0].min := 1.0, [1399].log_data[0].max := 1.0, [1399].log_data[0].total := 300.0, [1399].log_data[0].time := 300.0, [1399].log_data[0].minminute := 5, [1399].log_data[0].maxminute := 5, [1399].log_data[0].valid := 1,
        [1399].log_data[1].valid := 1, [1399].log_data[2].valid := 1, [1399].log_data[3].valid := 1, [1399].log_data[4].valid := 1, [1399].time.Year := 2022, [1399].time.Month := 4, [1399].time.Day := 28, [1399].time.Hour := 18, [1399].time.Minute := 9, [1399].time.Second := 59, [1399].time.DST_ON := 1, [1400].log_data[0].min := 1.0, [1400].log_data[0].max := 1.0, [1400].log_data[0].total := 300.0, [1400].log_data[0].time := 300.0, [1400].log_data[0].minminute := 10, [1400].log_data[0].maxminute := 10, [1400].log_data[0].valid := 1, [1400].log_data[1].valid := 1, [1400].log_data[2].valid := 1, [1400].log_data[3].valid := 1, [1400].log_data[4].valid := 1, [1400].time.Year := 2022, [1400].time.Month := 4, [1400].time.Day := 28, [1400].time.Hour := 18, [1400].time.Minute := 14, [1400].time.Second := 59, [1400].time.DST_ON := 1, [1401].log_data[0].min := 1.0, [1401].log_data[0].max := 1.0, [1401].log_data[0].total := 300.0, [1401].log_data[0].time := 300.0, [1401].log_data[0].minminute := 15, [1401].log_data[0].maxminute := 15, [1401].log_data[0].valid := 1, [1401].log_data[1].valid := 1, [1401].log_data[2].valid := 1, [1401].log_data[3].valid := 1, [1401].log_data[4].valid := 1, [1401].time.Year := 2022, [1401].time.Month := 4, [1401].time.Day := 28, [1401].time.Hour := 18, [1401].time.Minute := 19, [1401].time.Second := 59, [1401].time.DST_ON := 1, [1402].log_data[0].min := 1.0, [1402].log_data[0].max := 1.0, [1402].log_data[0].total := 300.0, [1402].log_data[0].time := 300.0, [1402].log_data[0].minminute := 20, [1402].log_data[0].maxminute := 20, [1402].log_data[0].valid := 1, [1402].log_data[1].valid := 1, [1402].log_data[2].valid := 1, [1402].log_data[3].valid := 1, [1402].log_data[4].valid := 1, [1402].time.Year := 2022, [1402].time.Month := 4,
        [1402].time.Day := 28, [1402].time.Hour := 18, [1402].time.Minute := 24, [1402].time.Second := 59, [1402].time.DST_ON := 1, [1403].log_data[0].min := 1.0, [1403].log_data[0].max := 1.0, [1403].log_data[0].total := 300.0, [1403].log_data[0].time := 300.0, [1403].log_data[0].minminute := 25, [1403].log_data[0].maxminute := 25, [1403].log_data[0].valid := 1, [1403].log_data[1].valid := 1, [1403].log_data[2].valid := 1, [1403].log_data[3].valid := 1, [1403].log_data[4].valid := 1, [1403].time.Year := 2022, [1403].time.Month := 4, [1403].time.Day := 28, [1403].time.Hour := 18, [1403].time.Minute := 29, [1403].time.Second := 59, [1403].time.DST_ON := 1, [1404].log_data[0].min := 1.0, [1404].log_data[0].max := 1.0, [1404].log_data[0].total := 300.0, [1404].log_data[0].time := 300.0, [1404].log_data[0].minminute := 30, [1404].log_data[0].maxminute := 30, [1404].log_data[0].valid := 1, [1404].log_data[1].valid := 1, [1404].log_data[2].valid := 1, [1404].log_data[3].valid := 1, [1404].log_data[4].valid := 1, [1404].time.Year := 2022, [1404].time.Month := 4, [1404].time.Day := 28, [1404].time.Hour := 18, [1404].time.Minute := 34, [1404].time.Second := 59, [1404].time.DST_ON := 1, [1405].log_data[0].min := 1.0, [1405].log_data[0].max := 1.0, [1405].log_data[0].total := 300.0, [1405].log_data[0].time := 300.0, [1405].log_data[0].minminute := 35, [1405].log_data[0].maxminute := 35, [1405].log_data[0].valid := 1, [1405].log_data[1].valid := 1, [1405].log_data[2].valid := 1, [1405].log_data[3].valid := 1, [1405].log_data[4].valid := 1, [1405].time.Year := 2022, [1405].time.Month := 4, [1405].time.Day := 28, [1405].time.Hour := 18, [1405].time.Minute := 39, [1405].time.Second := 59, [1405].time.DST_ON := 1, [1406].log_data[0].min := 1.0,
        [1406].log_data[0].max := 1.0, [1406].log_data[0].total := 300.0, [1406].log_data[0].time := 300.0, [1406].log_data[0].minminute := 40, [1406].log_data[0].maxminute := 40, [1406].log_data[0].valid := 1, [1406].log_data[1].valid := 1, [1406].log_data[2].valid := 1, [1406].log_data[3].valid := 1, [1406].log_data[4].valid := 1, [1406].time.Year := 2022, [1406].time.Month := 4, [1406].time.Day := 28, [1406].time.Hour := 18, [1406].time.Minute := 44, [1406].time.Second := 59, [1406].time.DST_ON := 1, [1407].log_data[0].min := 1.0, [1407].log_data[0].max := 1.0, [1407].log_data[0].total := 300.0, [1407].log_data[0].time := 300.0, [1407].log_data[0].minminute := 45, [1407].log_data[0].maxminute := 45, [1407].log_data[0].valid := 1, [1407].log_data[1].valid := 1, [1407].log_data[2].valid := 1, [1407].log_data[3].valid := 1, [1407].log_data[4].valid := 1, [1407].time.Year := 2022, [1407].time.Month := 4, [1407].time.Day := 28, [1407].time.Hour := 18, [1407].time.Minute := 49, [1407].time.Second := 59, [1407].time.DST_ON := 1, [1408].log_data[0].min := 1.0, [1408].log_data[0].max := 1.0, [1408].log_data[0].total := 300.0, [1408].log_data[0].time := 300.0, [1408].log_data[0].minminute := 50, [1408].log_data[0].maxminute := 50, [1408].log_data[0].valid := 1, [1408].log_data[1].valid := 1, [1408].log_data[2].valid := 1, [1408].log_data[3].valid := 1, [1408].log_data[4].valid := 1, [1408].time.Year := 2022, [1408].time.Month := 4, [1408].time.Day := 28, [1408].time.Hour := 18, [1408].time.Minute := 54, [1408].time.Second := 59, [1408].time.DST_ON := 1, [1409].log_data[0].min := 1.0, [1409].log_data[0].max := 1.0, [1409].log_data[0].total := 300.0, [1409].log_data[0].time := 300.0, [1409].log_data[0].minminute := 55, [1409].log_data[0].maxminute := 55, [1409].log_data[0].valid := 1,
        [1409].log_data[1].valid := 1, [1409].log_data[2].valid := 1, [1409].log_data[3].valid := 1, [1409].log_data[4].valid := 1, [1409].time.Year := 2022, [1409].time.Month := 4, [1409].time.Day := 28, [1409].time.Hour := 18, [1409].time.Minute := 59, [1409].time.Second := 59, [1409].time.DST_ON := 1, [1410].log_data[0].min := 1.0, [1410].log_data[0].max := 1.0, [1410].log_data[0].total := 300.0, [1410].log_data[0].time := 300.0, [1410].log_data[0].valid := 1, [1410].log_data[1].valid := 1, [1410].log_data[2].valid := 1, [1410].log_data[3].valid := 1, [1410].log_data[4].valid := 1, [1410].time.Year := 2022, [1410].time.Month := 4, [1410].time.Day := 28, [1410].time.Hour := 19, [1410].time.Minute := 4, [1410].time.Second := 59, [1410].time.DST_ON := 1, [1411].log_data[0].min := 1.0, [1411].log_data[0].max := 1.0, [1411].log_data[0].total := 300.0, [1411].log_data[0].time := 300.0, [1411].log_data[0].minminute := 5, [1411].log_data[0].maxminute := 5, [1411].log_data[0].valid := 1, [1411].log_data[1].valid := 1, [1411].log_data[2].valid := 1, [1411].log_data[3].valid := 1, [1411].log_data[4].valid := 1, [1411].time.Year := 2022, [1411].time.Month := 4, [1411].time.Day := 28, [1411].time.Hour := 19, [1411].time.Minute := 9, [1411].time.Second := 59, [1411].time.DST_ON := 1, [1412].log_data[0].min := 1.0, [1412].log_data[0].max := 1.0, [1412].log_data[0].total := 300.0, [1412].log_data[0].time := 300.0, [1412].log_data[0].minminute := 10, [1412].log_data[0].maxminute := 10, [1412].log_data[0].valid := 1, [1412].log_data[1].valid := 1, [1412].log_data[2].valid := 1, [1412].log_data[3].valid := 1, [1412].log_data[4].valid := 1, [1412].time.Year := 2022, [1412].time.Month := 4, [1412].time.Day := 28, [1412].time.Hour := 19,
        [1412].time.Minute := 14, [1412].time.Second := 59, [1412].time.DST_ON := 1, [1413].log_data[0].min := 1.0, [1413].log_data[0].max := 1.0, [1413].log_data[0].total := 300.0, [1413].log_data[0].time := 300.0, [1413].log_data[0].minminute := 15, [1413].log_data[0].maxminute := 15, [1413].log_data[0].valid := 1, [1413].log_data[1].valid := 1, [1413].log_data[2].valid := 1, [1413].log_data[3].valid := 1, [1413].log_data[4].valid := 1, [1413].time.Year := 2022, [1413].time.Month := 4, [1413].time.Day := 28, [1413].time.Hour := 19, [1413].time.Minute := 19, [1413].time.Second := 59, [1413].time.DST_ON := 1, [1414].log_data[0].min := 1.0, [1414].log_data[0].max := 1.0, [1414].log_data[0].total := 300.0, [1414].log_data[0].time := 300.0, [1414].log_data[0].minminute := 20, [1414].log_data[0].maxminute := 20, [1414].log_data[0].valid := 1, [1414].log_data[1].valid := 1, [1414].log_data[2].valid := 1, [1414].log_data[3].valid := 1, [1414].log_data[4].valid := 1, [1414].time.Year := 2022, [1414].time.Month := 4, [1414].time.Day := 28, [1414].time.Hour := 19, [1414].time.Minute := 24, [1414].time.Second := 59, [1414].time.DST_ON := 1, [1415].log_data[0].min := 1.0, [1415].log_data[0].max := 1.0, [1415].log_data[0].total := 300.0, [1415].log_data[0].time := 300.0, [1415].log_data[0].minminute := 25, [1415].log_data[0].maxminute := 25, [1415].log_data[0].valid := 1, [1415].log_data[1].valid := 1, [1415].log_data[2].valid := 1, [1415].log_data[3].valid := 1, [1415].log_data[4].valid := 1, [1415].time.Year := 2022, [1415].time.Month := 4, [1415].time.Day := 28, [1415].time.Hour := 19, [1415].time.Minute := 29, [1415].time.Second := 59, [1415].time.DST_ON := 1, [1416].log_data[0].min := 1.0, [1416].log_data[0].max := 1.0, [1416].log_data[0].total := 300.0,
        [1416].log_data[0].time := 300.0, [1416].log_data[0].minminute := 30, [1416].log_data[0].maxminute := 30, [1416].log_data[0].valid := 1, [1416].log_data[1].valid := 1, [1416].log_data[2].valid := 1, [1416].log_data[3].valid := 1, [1416].log_data[4].valid := 1, [1416].time.Year := 2022, [1416].time.Month := 4, [1416].time.Day := 28, [1416].time.Hour := 19, [1416].time.Minute := 34, [1416].time.Second := 59, [1416].time.DST_ON := 1, [1417].log_data[0].min := 1.0, [1417].log_data[0].max := 1.0, [1417].log_data[0].total := 300.0, [1417].log_data[0].time := 300.0, [1417].log_data[0].minminute := 35, [1417].log_data[0].maxminute := 35, [1417].log_data[0].valid := 1, [1417].log_data[1].valid := 1, [1417].log_data[2].valid := 1, [1417].log_data[3].valid := 1, [1417].log_data[4].valid := 1, [1417].time.Year := 2022, [1417].time.Month := 4, [1417].time.Day := 28, [1417].time.Hour := 19, [1417].time.Minute := 39, [1417].time.Second := 59, [1417].time.DST_ON := 1, [1418].log_data[0].min := 1.0, [1418].log_data[0].max := 1.0, [1418].log_data[0].total := 300.0, [1418].log_data[0].time := 300.0, [1418].log_data[0].minminute := 40, [1418].log_data[0].maxminute := 40, [1418].log_data[0].valid := 1, [1418].log_data[1].valid := 1, [1418].log_data[2].valid := 1, [1418].log_data[3].valid := 1, [1418].log_data[4].valid := 1, [1418].time.Year := 2022, [1418].time.Month := 4, [1418].time.Day := 28, [1418].time.Hour := 19, [1418].time.Minute := 44, [1418].time.Second := 59, [1418].time.DST_ON := 1, [1419].log_data[0].min := 1.0, [1419].log_data[0].max := 1.0, [1419].log_data[0].total := 300.0, [1419].log_data[0].time := 300.0, [1419].log_data[0].minminute := 45, [1419].log_data[0].maxminute := 45, [1419].log_data[0].valid := 1, [1419].log_data[1].valid := 1, [1419].log_data[2].valid := 1,
        [1419].log_data[3].valid := 1, [1419].log_data[4].valid := 1, [1419].time.Year := 2022, [1419].time.Month := 4, [1419].time.Day := 28, [1419].time.Hour := 19, [1419].time.Minute := 49, [1419].time.Second := 59, [1419].time.DST_ON := 1, [1420].log_data[0].min := 1.0, [1420].log_data[0].max := 1.0, [1420].log_data[0].total := 300.0, [1420].log_data[0].time := 300.0, [1420].log_data[0].minminute := 50, [1420].log_data[0].maxminute := 50, [1420].log_data[0].valid := 1, [1420].log_data[1].valid := 1, [1420].log_data[2].valid := 1, [1420].log_data[3].valid := 1, [1420].log_data[4].valid := 1, [1420].time.Year := 2022, [1420].time.Month := 4, [1420].time.Day := 28, [1420].time.Hour := 19, [1420].time.Minute := 54, [1420].time.Second := 59, [1420].time.DST_ON := 1, [1421].log_data[0].min := 1.0, [1421].log_data[0].max := 1.0, [1421].log_data[0].total := 300.0, [1421].log_data[0].time := 300.0, [1421].log_data[0].minminute := 55, [1421].log_data[0].maxminute := 55, [1421].log_data[0].valid := 1, [1421].log_data[1].valid := 1, [1421].log_data[2].valid := 1, [1421].log_data[3].valid := 1, [1421].log_data[4].valid := 1, [1421].time.Year := 2022, [1421].time.Month := 4, [1421].time.Day := 28, [1421].time.Hour := 19, [1421].time.Minute := 59, [1421].time.Second := 59, [1421].time.DST_ON := 1, [1422].log_data[0].min := 1.0, [1422].log_data[0].max := 1.0, [1422].log_data[0].total := 300.0, [1422].log_data[0].time := 300.0, [1422].log_data[0].valid := 1, [1422].log_data[1].valid := 1, [1422].log_data[2].valid := 1, [1422].log_data[3].valid := 1, [1422].log_data[4].valid := 1, [1422].time.Year := 2022, [1422].time.Month := 4, [1422].time.Day := 28, [1422].time.Hour := 20, [1422].time.Minute := 4, [1422].time.Second := 59,
        [1422].time.DST_ON := 1, [1423].log_data[0].min := 1.0, [1423].log_data[0].max := 1.0, [1423].log_data[0].total := 300.0, [1423].log_data[0].time := 300.0, [1423].log_data[0].minminute := 5, [1423].log_data[0].maxminute := 5, [1423].log_data[0].valid := 1, [1423].log_data[1].valid := 1, [1423].log_data[2].valid := 1, [1423].log_data[3].valid := 1, [1423].log_data[4].valid := 1, [1423].time.Year := 2022, [1423].time.Month := 4, [1423].time.Day := 28, [1423].time.Hour := 20, [1423].time.Minute := 9, [1423].time.Second := 59, [1423].time.DST_ON := 1, [1424].log_data[0].min := 1.0, [1424].log_data[0].max := 1.0, [1424].log_data[0].total := 300.0, [1424].log_data[0].time := 300.0, [1424].log_data[0].minminute := 10, [1424].log_data[0].maxminute := 10, [1424].log_data[0].valid := 1, [1424].log_data[1].valid := 1, [1424].log_data[2].valid := 1, [1424].log_data[3].valid := 1, [1424].log_data[4].valid := 1, [1424].time.Year := 2022, [1424].time.Month := 4, [1424].time.Day := 28, [1424].time.Hour := 20, [1424].time.Minute := 14, [1424].time.Second := 59, [1424].time.DST_ON := 1, [1425].log_data[0].min := 1.0, [1425].log_data[0].max := 1.0, [1425].log_data[0].total := 300.0, [1425].log_data[0].time := 300.0, [1425].log_data[0].minminute := 15, [1425].log_data[0].maxminute := 15, [1425].log_data[0].valid := 1, [1425].log_data[1].valid := 1, [1425].log_data[2].valid := 1, [1425].log_data[3].valid := 1, [1425].log_data[4].valid := 1, [1425].time.Year := 2022, [1425].time.Month := 4, [1425].time.Day := 28, [1425].time.Hour := 20, [1425].time.Minute := 19, [1425].time.Second := 59, [1425].time.DST_ON := 1, [1426].log_data[0].min := 1.0, [1426].log_data[0].max := 1.0, [1426].log_data[0].total := 300.0, [1426].log_data[0].time := 300.0, [1426].log_data[0].minminute := 20,
        [1426].log_data[0].maxminute := 20, [1426].log_data[0].valid := 1, [1426].log_data[1].valid := 1, [1426].log_data[2].valid := 1, [1426].log_data[3].valid := 1, [1426].log_data[4].valid := 1, [1426].time.Year := 2022, [1426].time.Month := 4, [1426].time.Day := 28, [1426].time.Hour := 20, [1426].time.Minute := 24, [1426].time.Second := 59, [1426].time.DST_ON := 1, [1427].log_data[0].min := 1.0, [1427].log_data[0].max := 1.0, [1427].log_data[0].total := 300.0, [1427].log_data[0].time := 300.0, [1427].log_data[0].minminute := 25, [1427].log_data[0].maxminute := 25, [1427].log_data[0].valid := 1, [1427].log_data[1].valid := 1, [1427].log_data[2].valid := 1, [1427].log_data[3].valid := 1, [1427].log_data[4].valid := 1, [1427].time.Year := 2022, [1427].time.Month := 4, [1427].time.Day := 28, [1427].time.Hour := 20, [1427].time.Minute := 29, [1427].time.Second := 59, [1427].time.DST_ON := 1, [1428].log_data[0].min := 1.0, [1428].log_data[0].max := 1.0, [1428].log_data[0].total := 300.0, [1428].log_data[0].time := 300.0, [1428].log_data[0].minminute := 30, [1428].log_data[0].maxminute := 30, [1428].log_data[0].valid := 1, [1428].log_data[1].valid := 1, [1428].log_data[2].valid := 1, [1428].log_data[3].valid := 1, [1428].log_data[4].valid := 1, [1428].time.Year := 2022, [1428].time.Month := 4, [1428].time.Day := 28, [1428].time.Hour := 20, [1428].time.Minute := 34, [1428].time.Second := 59, [1428].time.DST_ON := 1, [1429].log_data[0].min := 1.0, [1429].log_data[0].max := 1.0, [1429].log_data[0].total := 300.0, [1429].log_data[0].time := 300.0, [1429].log_data[0].minminute := 35, [1429].log_data[0].maxminute := 35, [1429].log_data[0].valid := 1, [1429].log_data[1].valid := 1, [1429].log_data[2].valid := 1, [1429].log_data[3].valid := 1, [1429].log_data[4].valid := 1,
